PROPERTY NumOfHangers : DINT
GET
NumOfHangers:= SIf.Cur.dinNumOfHangersInBuffer;
END_GET
END_PROPERTY

METHOD PROTECTED sta_ERROR : BOOL
// state implemetation
//--------------------------------------------------------------------------------------
// Entry action
	IF (me.StateMachine.intState<>me.StateMachine.intStateLastCycle) THEN
		me.StateMachine.intStateHistory := me.StateMachine.intStateLastCycle; // -> possibillity to go back to state before error
		me.StateMachine.intStateLastCycle := me.StateMachine.intState;
		
	END_IF

//--------------------------------------------------------------------------------------
// Cyclic action
	IF (me.StateMachine.intState=me.StateMachine.intStateLastCycle) THEN
		
		// Switch valve off, cylinder back to extend position -> stop hanger
		SIf.Out.bolRetract.intern := FALSE;
		SIf.Out.bolRetract2.intern := TRUE;	
		
		// State Change Condition
		IF (CIf.Job.bolAlmReset = TRUE) THEN
			me.StateMachine.intStateNext := cSTA_ERRORQuit;
		END_IF
	END_IF

//--------------------------------------------------------------------------------------
// Exit action
	IF (me.StateMachine.intState<>me.StateMachine.intStateNext) THEN
		;
	END_IF
END_METHOD

METHOD PROTECTED sta_OFF : BOOL
// state implemetation
//--------------------------------------------------------------------------------------
// Entry action
	IF (me.StateMachine.intState<>me.StateMachine.intStateLastCycle) THEN
		me.StateMachine.intStateLastCycle := me.StateMachine.intState;
		
		// Reset total counter
		SIf.Cur.dinHangersPassedTotal:= 0;
	END_IF


//--------------------------------------------------------------------------------------
// Cyclic action
	IF (me.StateMachine.intState=me.StateMachine.intStateLastCycle) THEN
		
	
		// State Change Condition
		IF (me.Alarm.eActivAlmClass<>E_AlmClass.EOFF) AND (me.Alarm.eActivAlmClass<>E_AlmClass.OFF) THEN
			IF (me.intCmd=cCMD_STOP) THEN
				me.StateMachine.intStateNext :=  cSTA_STOPBusy;
			ELSIF (me.intCmd=STB_CmdState.cCMD_RELEASE) THEN 
				me.StateMachine.intStateNext := STB_CmdState.cSTA_RELEASEBusy;
			ELSIF(me.intCmd=STB_CmdState.cCMD_RELEASE_ALL) THEN
				me.StateMachine.intStateNext := STB_CmdState.cSTA_RELEASE_ALLBusy;
			ELSIF(me.intCmd=cCMD_RUN) THEN
				me.StateMachine.intStateNext := cSTA_RUNBusy;
			END_IF
		END_IF
	END_IF


//--------------------------------------------------------------------------------------
// Exit action
	IF (me.StateMachine.intState<>me.StateMachine.intStateNext) THEN
		;
	END_IF
END_METHOD

METHOD PROTECTED sta_OFFBusy : BOOL
// state implemetation
//--------------------------------------------------------------------------------------
// Entry action
	IF (me.StateMachine.intState<>me.StateMachine.intStateLastCycle) THEN
		me.StateMachine.intStateLastCycle := me.StateMachine.intState;
			
	END_IF

//--------------------------------------------------------------------------------------
// Cyclic action
	IF (me.StateMachine.intState=me.StateMachine.intStateLastCycle) THEN
		
		// Switch valve off, cylinder back to extend position -> stop hanger
		SIf.Out.bolRetract.intern := FALSE;
		SIf.Out.bolRetract2.intern := TRUE;	
			
		// State Change Condition
		IF (FALSE) THEN
			;
		ELSIF (TRUE) THEN
			me.StateMachine.intStateNext := cSTA_OFF;
		END_IF
	END_IF


//--------------------------------------------------------------------------------------
// Exit action
	IF (me.StateMachine.intState<>me.StateMachine.intStateNext) THEN
		;
	END_IF
END_METHOD

METHOD PROTECTED sta_RELEASE : BOOL
// state implemetation
//--------------------------------------------------------------------------------------
// Entry action
	IF (me.StateMachine.intState<>me.StateMachine.intStateLastCycle) THEN
		me.StateMachine.intStateLastCycle := me.StateMachine.intState;
			
		;
	END_IF

//--------------------------------------------------------------------------------------
// Cyclic action
	IF (me.StateMachine.intState=me.StateMachine.intStateLastCycle) THEN
		
		// Switch valve off, cylinder back to extend position -> stop hanger
		SIf.Out.bolRetract.intern := FALSE;
		SIf.Out.bolRetract2.intern := TRUE;	
		
		// State Change Condition
		IF (me.intCmd=cCMD_STOP) THEN
			me.StateMachine.intStateNext := cSTA_STOPBusy;
		ELSIF(me.intCmd=STB_CmdState.cCMD_RELEASE_ALL) THEN
			me.StateMachine.intStateNext := STB_CmdState.cSTA_RELEASE_ALLBusy;
		END_IF
		
	END_IF

//--------------------------------------------------------------------------------------
// Exit action
	IF (me.StateMachine.intState<>me.StateMachine.intStateNext) THEN
		;
	END_IF
END_METHOD

METHOD PROTECTED sta_RELEASE_ALL : BOOL
// state implemetation
//--------------------------------------------------------------------------------------
// Entry action
	IF (me.StateMachine.intState<>me.StateMachine.intStateLastCycle) THEN
		me.StateMachine.intStateLastCycle := me.StateMachine.intState;	
		;
	END_IF

//--------------------------------------------------------------------------------------
// Cyclic action
	IF (me.StateMachine.intState=me.StateMachine.intStateLastCycle) THEN
		

		// State Change Condition
		IF ((me.intCmd=cCMD_STOP) OR (me.intCmd=STB_CmdState.cCMD_RELEASE)) THEN
			me.StateMachine.intStateNext := cSTA_STOPBusy;
		END_IF
	END_IF

//--------------------------------------------------------------------------------------
// Exit action
	IF (me.StateMachine.intState<>me.StateMachine.intStateNext) THEN
		;
	END_IF
END_METHOD

METHOD PROTECTED sta_RELEASE_ALLBusy : BOOL
// state implemetation
//--------------------------------------------------------------------------------------
// Entry action
	IF (me.StateMachine.intState<>me.StateMachine.intStateLastCycle) THEN
		me.StateMachine.intStateLastCycle := me.StateMachine.intState;
				
		dinNumOfHangersToRelease:= 0;
		dinSetNumOfHangersToRelease:= 0;
		
		// Reset package counter
		SIf.Cur.dinHangersPassedPackage:= 0;
	
		// Initialize sub state machine
		me.SubStateMachine.intState:= cSTA_SUB_INITIALIZED; 
		me.SubStateMachine.intStateNext:= cSTA_SUB_INITIALIZED;
	
	END_IF

//--------------------------------------------------------------------------------------
// Cyclic action
	IF (me.StateMachine.intState=me.StateMachine.intStateLastCycle) THEN
			
		//--------------------------------------------------------------------------------------
		// sub state machine for release all sequence
		CASE me.SubStateMachine.intState OF
			//--------------------------------------------------------------------------------------
			cSTA_SUB_INITIALIZED:
				// Entry action
				IF (me.SubStateMachine.intState<>me.SubStateMachine.intStateLastCycle) THEN
					me.SubStateMachine.intStateLastCycle := me.SubStateMachine.intState;							
					
					//Used buffer mode?
					CASE SIf.Par.usiBuffermode OF
					0: // 0= Emptying buffer, use buffer capacity at cycle start
						dinSetNumOfHangersToRelease := SIf.Cfg.dinMaxCapacity;
					1: // 1= Emptying buffer, newly added hangers will be considered
						dinSetNumOfHangersToRelease := dinNumOfHangersToRelease;
					END_CASE
				
				END_IF
				
				// Simulation
				IF (CIf.SwCfg.bolSimulation) THEN
					;
				END_IF
	
				// State Change Condition
				IF(TRUE)THEN
					me.SubStateMachine.intStateNext := cSTA_SUB_HANGER_PASSING;
				END_IF
						
			//--------------------------------------------------------------------------------------
			cSTA_SUB_HANGER_PASSING:
				// Entry action
				IF (me.SubStateMachine.intState<>me.SubStateMachine.intStateLastCycle) THEN
					me.SubStateMachine.intStateLastCycle := me.SubStateMachine.intState;							
									
					// Check if min. one hanger exist and save info tmp. Used for counting.
					IF (SIf.In.bolHangerDetected.intern = TRUE) THEN
						bolHangerDetected:= TRUE;
					ELSE
						bolHangerDetected:= FALSE;
					END_IF
					
				END_IF
				
				// Simulation
				IF (CIf.SwCfg.bolSimulation) THEN
					;
				END_IF

				// Release all based on time and both pins go up or with pulses
				IF (SIf.Cfg.bolReleaseAllNonPulse = TRUE) THEN
					
					SIf.Out.bolRetract.intern := TRUE; // both pins move up
					SIf.Out.bolRetract2.intern := TRUE; // both pins move up
					
					// wait release all time
					IF (me.SubStateMachine.udiTimeInState_ms > SIf.Par.udiReleaseAllTime_ms) THEN
						me.SubStateMachine.intStateNext := cSTA_SUB_HANGER_PASSED;
					END_IF
					
					// Calculate number of hangers in buffer dependent number of hangers per pulse
					SIf.Cur.dinNumOfHangersInBuffer := 0;
					// Calculate total counter dependent number of hangers per pulse
					SIf.Cur.dinHangersPassedTotal:= SIf.Cur.dinHangersPassedTotal + dinNumOfHangersToRelease;
					// Calculate package counter dependent number of hangers per pulse				
					SIf.Cur.dinHangersPassedPackage:= SIf.Cur.dinHangersPassedPackage + dinNumOfHangersToRelease;
					// calculate hangers still to release
					dinSetNumOfHangersToRelease := 0;
					
				ELSE
					
					// Switch valve on, cylinder to retract position -> release hanger
					SIf.Out.bolRetract.intern := TRUE;  // pin move up
					SIf.Out.bolRetract2.intern := FALSE;  // pin move down
					
					// Pulse timer expired?
					IF (me.SubStateMachine.udiTimeInState_ms > SIf.Par.udiPulseLengthValve_ms) THEN
						me.SubStateMachine.intStateNext := cSTA_SUB_HANGER_PASSED;
						
						// Update all counters. Only if a hanger was detected before.
						// If no hanger detection sensor exists, count unconditional with every cylinder stroke
						IF (bolHangerDetected = TRUE) OR (Sif.Cfg.bolHasHangerDetection = FALSE) THEN
							
							// Note: Only for separator the number of hangers per pulse corresponds exactly the real number of passed hangers.
							// For all other units like e.g. double stopper it's only an approximate number.
						
							IF (SIf.Cfg.bolHasDecrementSensor = FALSE) THEN // Else do it in Method Always
								// Calculate number of hangers in buffer dependent number of hangers per pulse
								SIf.Cur.dinNumOfHangersInBuffer:= SIf.Cur.dinNumOfHangersInBuffer - dinNumOfHangersToRelease;
							END_IF
							// Calculate total counter dependent number of hangers per pulse
							SIf.Cur.dinHangersPassedTotal:= SIf.Cur.dinHangersPassedTotal + dinNumOfHangersToRelease;
							// Calculate package counter dependent number of hangers per pulse				
							SIf.Cur.dinHangersPassedPackage:= SIf.Cur.dinHangersPassedPackage + dinNumOfHangersToRelease;
							// calculate hangers still to release
							dinSetNumOfHangersToRelease := dinSetNumOfHangersToRelease - dinNumOfHangersToRelease;
							
							// Calculate NumOfHangersToRelease, Used for RELEASE_ALL end condition
							// Has buffer?
							// calculate max number of hangers could release per pulse
							IF (SIf.Cur.dinNumOfHangersInBuffer<=SIf.Cfg.uinNumOfHangersPerPulse) THEN
								dinNumOfHangersToRelease := SIf.Cur.dinNumOfHangersInBuffer;
							ELSE
								dinNumOfHangersToRelease := SIf.Cfg.uinNumOfHangersPerPulse;
							END_IF
							
							//Used buffer mode?
							CASE SIf.Par.usiBuffermode OF
								0:  
									IF  (dinNumOfHangersToRelease <= 0) THEN // All hangers should be released, do the hole capacity 
										dinSetNumOfHangersToRelease:= dinSetNumOfHangersToRelease - SIf.Cfg.uinNumOfHangersPerPulse;
									END_IF
								1:
									dinSetNumOfHangersToRelease:= dinNumOfHangersToRelease;
							END_CASE
													
							bolHangerDetected:= FALSE;
						END_IF
					END_IF
						
				END_IF
	
			//--------------------------------------------------------------------------------------
			cSTA_SUB_HANGER_PASSED:
				// Entry action
				IF (me.SubStateMachine.intState<>me.SubStateMachine.intStateLastCycle) THEN
					me.SubStateMachine.intStateLastCycle := me.SubStateMachine.intState;							
					;						
				END_IF
				
				// Switch valve off, cylinder back to extend position -> stop hanger
				SIf.Out.bolRetract.intern := FALSE;
				SIf.Out.bolRetract2.intern := TRUE;	
				
				// Simulation
				IF (CIf.SwCfg.bolSimulation) THEN
					;
				END_IF
					
				// State Change Condition
				IF ((dinSetNumOfHangersToRelease<=0) AND ((Sif.Cfg.bolHasHangerDetection = FALSE) OR (SIf.Par.usiBuffermode<>1))) THEN
					me.SubStateMachine.intStateNext := cSTA_SUB_FINISHED;
				ELSIF ((SIf.Par.usiBuffermode=1) AND (Sif.Cfg.bolHasHangerDetection = TRUE) AND (SIf.In.bolHangerDetected.intern = FALSE)) THEN
					me.SubStateMachine.intStateNext := cSTA_SUB_FINISHED;
				ELSIF (me.SubStateMachine.udiTimeInState_ms > SIf.Par.udiIntervalBufferEmptying_ms) THEN
					me.SubStateMachine.intStateNext := cSTA_SUB_HANGER_PASSING;
				END_IF
			
			//--------------------------------------------------------------------------------------
			cSTA_SUB_FINISHED:
					;	// Buffer emptied 
					
		END_CASE
			
		// State Change Condition
		// [ms] Timeout buffer emptying -> ERROR,(0 = disable monitoring)
		IF ((me.StateMachine.udiTimeInState_ms > (SIf.Par.udiTimeoutBufferEmptying_ms)) AND (SIf.Par.udiTimeoutBufferEmptying_ms <> 0)) THEN
			// SIf.Alm[1].strText := 'Timeout buffer emptying';
			pfbAlarmCtrl^.setAlarm(CIf.Info.intCtrlId,1,0,ADR(SIf.Alm),E_AlmState.RST,CIf.Job.eMe_ActivAlmClass);
			me.StateMachine.intStateNext := cSTA_ERROR;
		ELSIF (me.SubStateMachine.intState = cSTA_SUB_FINISHED) THEN				// Buffer emptied -> RELEASE_ALL
			me.StateMachine.intStateNext := STB_CmdState.cSTA_RELEASE_ALL;
		ELSIF(me.intCmd=cCMD_STOP) THEN
			me.StateMachine.intStateNext := cSTA_STOPBusy;		
		END_IF
	END_IF


//--------------------------------------------------------------------------------------
// Exit action
	IF (me.StateMachine.intState<>me.StateMachine.intStateNext) THEN
		;
	END_IF
END_METHOD

METHOD PROTECTED sta_RELEASEBusy : BOOL
// state implemetation
//--------------------------------------------------------------------------------------
// Entry action
	IF (me.StateMachine.intState<>me.StateMachine.intStateLastCycle) THEN
		me.StateMachine.intStateLastCycle := me.StateMachine.intState;

		// Check if min. one hanger exist and save info tmp. Used for counting in state RELEASE.	
		IF (SIf.In.bolHangerDetected.intern = TRUE) THEN
			bolHangerDetected:= TRUE;
		ELSE
			bolHangerDetected:= FALSE;
		END_IF
	
	END_IF

//--------------------------------------------------------------------------------------
// Cyclic action
	IF (me.StateMachine.intState=me.StateMachine.intStateLastCycle) THEN
		
		// Switch valve on, cylinder to retract position -> release hanger
		SIf.Out.bolRetract.intern := TRUE;
		SIf.Out.bolRetract2.intern := FALSE;	
		
		// State Change Condition
		IF (me.StateMachine.udiTimeInState_ms > SIf.Par.udiPulseLengthValve_ms) THEN
			me.StateMachine.intStateNext := STB_CmdState.cSTA_RELEASE;
	
			// Update all counters. Only if a hanger was detected before.
			// If no hanger detection sensor exists, count unconditional with every cylinder stroke
			IF (bolHangerDetected = TRUE) OR (SIf.Cfg.bolHasHangerDetection = FALSE) THEN
				
				// Note: Only for separator the number of hangers per pulse corresponds exactly the real number of passed hangers.
				// For all other units like e.g. double stopper it's only an approximate number.
			
				IF (SIf.Cfg.bolHasDecrementSensor = FALSE) THEN // Else do it in Method Always
					IF (SIf.Cfg.bolHasBufferFullSensor = TRUE AND SIf.In.bolBufferFull.intern = FALSE) THEN
						// Calculate number of hangers in buffer dependent number of hangers per pulse
						SIf.Cur.dinNumOfHangersInBuffer:= SIf.Cur.dinNumOfHangersInBuffer - dinNumOfHangersToRelease;
					ELSIF SIf.Cfg.bolHasBufferFullSensor = FALSE THEN
						// Calculate number of hangers in buffer dependent number of hangers per pulse
						SIf.Cur.dinNumOfHangersInBuffer:= SIf.Cur.dinNumOfHangersInBuffer - dinNumOfHangersToRelease;						
					END_IF
				END_IF
					
				// Calculate total counter dependent number of hangers per pulse
				SIf.Cur.dinHangersPassedTotal:= SIf.Cur.dinHangersPassedTotal + dinNumOfHangersToRelease;
				
				bolHangerDetected:= FALSE;
			END_IF
				
		END_IF
		
	END_IF

//--------------------------------------------------------------------------------------
// Exit action
	IF (me.StateMachine.intState<>me.StateMachine.intStateNext) THEN
		;
	END_IF
END_METHOD

METHOD PROTECTED sta_RUN : BOOL
// state implemetation
//--------------------------------------------------------------------------------------
// Entry action
	IF (me.StateMachine.intState<>me.StateMachine.intStateLastCycle) THEN
		me.StateMachine.intStateLastCycle := me.StateMachine.intState;
		
		// Init sub state machine	
		me.SubStateMachine.intState := cSTA_SUB_CHECK_FOR_RESERVATION; 
		me.SubStateMachine.intStateNext := cSTA_SUB_CHECK_FOR_RESERVATION; 
	END_IF

//--------------------------------------------------------------------------------------
// Cyclic action
	IF (me.StateMachine.intState=me.StateMachine.intStateLastCycle) THEN
		
		//----------------------------------------------------------------------
		// Calculate position for transport 
		//----------------------------------------------------------------------	
		// If this task is in faster cycle then the parent, calculate internal position more exactly during the taskcycle
		IF dinTransportPositionOld_um <> SIf.Cur.dinTransportPosition_um THEN
			SIf.Cur.dinTransportPositionCalc_um := SIf.Cur.dinTransportPosition_um;
			dinTransportPositionOld_um := SIf.Cur.dinTransportPosition_um;
			dinPositionCorrection_um := 0;
		ELSE
			dinPositionCorrection_um := dinPositionCorrection_um + LREAL_TO_DINT(DINT_TO_LREAL(SIf.Cur.dinTransportspeed_um_s) * UDINT_TO_LREAL(me.FUBInfo.udiSample_ms) / 1000.0 );
			SIf.Cur.dinTransportPositionCalc_um := dinTransportPositionOld_um + dinPositionCorrection_um;
		END_IF
				
		//--------------------------------------------------------------------------------------
		// sub state machine
		CASE me.SubStateMachine.intState OF
			//--------------------------------------------------------------------------------------
			cSTA_SUB_CHECK_FOR_RESERVATION:
			
				IF (me.SubStateMachine.intState<>me.SubStateMachine.intStateLastCycle) THEN
					me.SubStateMachine.intStateLastCycle := me.SubStateMachine.intState;
					;
				END_IF
			
				// Simulation
				IF (CIf.SwCfg.bolSimulation) THEN
					;
				END_IF
							
				// Calculate trigger "negative" position offset.
				// Note: The trigger offset must be calculated dependent the drive (transport) speed 
				// Formular: TrigNegPosOffset = DriveSpeed * TimeOnSlide	
				dinCalcTrigNegPosOffset_um:= REAL_TO_DINT (DINT_TO_REAL(SIf.Cur.dinTransportspeed_um_s) * (UINT_TO_REAL(SIf.Par.uinTimeOnSlide_ms) / 1000));
					
				// Check trigger window
				FOR intBufferIndex := 0 TO Const_MTR.cusiSectionBuffer_SIZE DO
					// Check if the current transport position is within the trigger window and if section is reserved for this instance to release the hanger
					IF ((SIf.Par.dinPositionOfSlide_um < (SIf.Cur.pSectionBuffer^[intBufferIndex].dinTrigStartPos - dinCalcTrigNegPosOffset_um))
						AND (SIf.Par.dinPositionOfSlide_um > (SIf.Cur.pSectionBuffer^[intBufferIndex].dinTrigEndPos - dinCalcTrigNegPosOffset_um))
						AND (SIf.Cur.pSectionBuffer^[intBufferIndex].enmState = E_Typ_MTR_SECTION_STATE.Reserved) AND (SIf.Cur.pSectionBuffer^[intBufferIndex].usiReservedForLine = SIf.Cfg.usiLineNumber)) THEN						
							// Section is free and reserved for this instance -> hanger can be released!
							// Update status for the section
							SIf.Cur.pSectionBuffer^[intBufferIndex].enmState := E_Typ_MTR_SECTION_STATE.HangerOnSlide;
							me.SubStateMachine.intStateNext := cSTA_SUB_RELEASE_BUSY;
							EXIT;
					END_IF
				END_FOR					
				
			//--------------------------------------------------------------------------------------
			cSTA_SUB_RELEASE_BUSY:
				IF (me.SubStateMachine.intState<>me.SubStateMachine.intStateLastCycle) THEN
					me.SubStateMachine.intStateLastCycle := me.SubStateMachine.intState;
					;
				END_IF
			
				// Switch valve on, cylinder to retract position -> release hanger
				SIf.Out.bolRetract.intern := TRUE;
				
				// State Change Condition
				IF (me.SubStateMachine.udiTimeInState_ms > SIf.Par.udiPulseLengthValve_ms) THEN
					// Next step
					me.SubStateMachine.intStateNext := cSTA_SUB_STOP;
			
					// Update all counters. Only if a hanger was detected before.
					// If no hanger detection sensor exists, count unconditional with every cylinder stroke
					IF (SIf.In.bolHangerDetected.intern = TRUE) OR (SIf.Cfg.bolHasHangerDetection = FALSE) THEN
						
						// Note: Only for separator the number of hangers per pulse corresponds exactly the real number of passed hangers.
						// For all other units like e.g. double stopper it's only an approximate number.
					
						IF (SIf.Cfg.bolHasDecrementSensor = FALSE) THEN // Else do it in Method Always
							IF (SIf.Cfg.bolHasBufferFullSensor = TRUE AND SIf.In.bolBufferFull.intern = FALSE) THEN
								// Calculate number of hangers in buffer dependent number of hangers per pulse
								SIf.Cur.dinNumOfHangersInBuffer:= SIf.Cur.dinNumOfHangersInBuffer - dinNumOfHangersToRelease;
							ELSIF SIf.Cfg.bolHasBufferFullSensor = FALSE THEN
								// Calculate number of hangers in buffer dependent number of hangers per pulse
								SIf.Cur.dinNumOfHangersInBuffer:= SIf.Cur.dinNumOfHangersInBuffer - dinNumOfHangersToRelease;						
							END_IF
						END_IF						
						// Calculate total counter dependent number of hangers per pulse
						SIf.Cur.dinHangersPassedTotal:= SIf.Cur.dinHangersPassedTotal + dinNumOfHangersToRelease;		
					END_IF
						
				END_IF
			
			//--------------------------------------------------------------------------------------
			cSTA_SUB_STOP:
				IF (me.SubStateMachine.intState<>me.SubStateMachine.intStateLastCycle) THEN
					me.SubStateMachine.intStateLastCycle := me.SubStateMachine.intState;
				END_IF
				
				// Update status for the section
				SIf.Cur.pSectionBuffer^[intBufferIndex].enmState := E_Typ_MTR_SECTION_STATE.HangerReleased;
				// Switch valve off, cylinder back to extend position -> stop hanger
				SIf.Out.bolRetract.intern := FALSE;
			
				// State Change Condition
				// Check error if retracted position not reached
				IF (TRUE) THEN
					me.SubStateMachine.intStateNext := cSTA_SUB_CHECK_FOR_RESERVATION;
				END_IF
		
			
		END_CASE
		
		// State Change Condition
		IF(me.intCmd=cCMD_STOP) THEN
			me.StateMachine.intStateNext := cSTA_STOPBusy;	
		END_IF
		
	END_IF

//--------------------------------------------------------------------------------------
// Exit action
	IF (me.StateMachine.intState<>me.StateMachine.intStateNext) THEN
	;
	END_IF
END_METHOD

METHOD PROTECTED sta_RUNBusy : BOOL
// state implemetation
//--------------------------------------------------------------------------------------
// Entry action
	IF (me.StateMachine.intState<>me.StateMachine.intStateLastCycle) THEN
		me.StateMachine.intStateLastCycle := me.StateMachine.intState;
		;				
	END_IF

//--------------------------------------------------------------------------------------
// Cyclic action
	IF (me.StateMachine.intState=me.StateMachine.intStateLastCycle) THEN
			
		// State Change Condition
		
		// Check if access to section buffer exist. 
		// This controller will be set to RUN in case if STB work in combination with FUB MTR to merge hangers into a TLK.
		IF (SIf.Cur.pSectionBuffer = 0) THEN
			// SIf.Alm[4].strText := 'RUN not possible, no access to section buffer';
			pfbAlarmCtrl^.setAlarm(CIf.Info.intCtrlId,4,0,ADR(SIf.Alm),E_AlmState.RST,CIf.Job.eMe_ActivAlmClass);	
			me.StateMachine.intStateNext := cSTA_ERROR;
		ELSE
			me.StateMachine.intStateNext := cSTA_RUN;		
		END_IF
	END_IF

//--------------------------------------------------------------------------------------
// Exit action
	IF (me.StateMachine.intState<>me.StateMachine.intStateNext) THEN
		;
	END_IF
END_METHOD

METHOD PROTECTED sta_STOP : BOOL
// state implemetation
//--------------------------------------------------------------------------------------
// Entry action
	IF (me.StateMachine.intState<>me.StateMachine.intStateLastCycle) THEN
		me.StateMachine.intStateLastCycle := me.StateMachine.intState;
		
		bolErrorPosLost:= FALSE;
		uinPosEdgeCounter:= 0;
	END_IF


//--------------------------------------------------------------------------------------
// Cyclic action
	IF (me.StateMachine.intState=me.StateMachine.intStateLastCycle) THEN
	
		//--------------------------------------------------------------------
		// Monitoring for cylinder position lost
		//--------------------------------------------------------------------
		IF (Sif.cfg.bolCylPosLostMonitoring=TRUE) THEN
			
			// -> Checked indirectly via sensor "buffer full" or "hanger detected" if exist.
			
			// Decision, which sensor should be used for monitoring
			// Prio 1. Always use the hanger detection sensor if exists
			IF (SIf.Cfg.bolHasHangerDetection = TRUE) THEN
				// Use hanger detection sensor signal
				bolSignalForPosLostMonitoring:= SIf.In.bolHangerDetected.intern;
			ELSE
				// Prio 2. Check if buffer full sensor exists 
				IF (SIf.Cfg.bolHasBufferFullSensor = TRUE) THEN
					// Use buffer full sensor signal
					bolSignalForPosLostMonitoring:= SIf.In.bolBufferFull.intern;
				ELSE
					// No sensor exist. Not possible to monitor cylinder position lost! 
					bolSignalForPosLostMonitoring:= FALSE;
				END_IF
			END_IF
				
			// Count sensor pos. edges
			IF ((bolSignalForPosLostMonitoring <> bolSignalForPosLostMonitoringOld) AND (bolSignalForPosLostMonitoring = TRUE))THEN	
				uinPosEdgeCounter:= uinPosEdgeCounter + 1;
			END_IF
			bolSignalForPosLostMonitoringOld:= bolSignalForPosLostMonitoring;
						
			// Check condition for set error
			// Wait until the counter is > than dinMaxNumOfHangers_PosMonitoring
			IF (uinPosEdgeCounter > SIf.Cfg.dinMaxNumOfHangers_PosMonitoring) THEN
				bolErrorPosLost:= TRUE;
			END_IF
			
		END_IF
		
		//--------------------------------------------------------------------
		//--------------------------------------------------------------------
		
		// State Change Condition	
		// Error cylinder position lost
		IF ((bolErrorPosLost=TRUE) AND (Sif.cfg.bolCylPosLostMonitoring=TRUE))THEN
			// SIf.Alm[3].strText := 'Cylinder position lost. Hangers slip through';
			pfbAlarmCtrl^.setAlarm(CIf.Info.intCtrlId,3,0,ADR(SIf.Alm),E_AlmState.RST,CIf.Job.eMe_ActivAlmClass);
			bolErrorPosLost:= FALSE;
			uinPosEdgeCounter:= 0;
			me.StateMachine.intStateNext := cSTA_ERROR;
		ELSIF (me.intCmd=STB_CmdState.cCMD_RELEASE) THEN 
			me.StateMachine.intStateNext := STB_CmdState.cSTA_RELEASEBusy;
		ELSIF(me.intCmd=STB_CmdState.cCMD_RELEASE_ALL) THEN
			me.StateMachine.intStateNext := STB_CmdState.cSTA_RELEASE_ALLBusy;
		ELSIF (me.intCmd=cCMD_RUN) THEN
			me.StateMachine.intStateNext := cSTA_RUNBusy;
		END_IF
	END_IF

//-------------------------------------------------------------------------------------
// Exit action
	IF (me.StateMachine.intState<>me.StateMachine.intStateNext) THEN
		;
	END_IF
END_METHOD

METHOD PROTECTED sta_STOPBusy : BOOL
// state implemetation
//--------------------------------------------------------------------------------------
// Entry action
	IF (me.StateMachine.intState<>me.StateMachine.intStateLastCycle) THEN
		me.StateMachine.intStateLastCycle := me.StateMachine.intState;

	END_IF


//--------------------------------------------------------------------------------------
// Cyclic action
	IF (me.StateMachine.intState=me.StateMachine.intStateLastCycle) THEN
			
		// Switch valve off, cylinder back to extend position -> stop hanger
		SIf.Out.bolRetract.intern := FALSE;
		SIf.Out.bolRetract2.intern := TRUE;	
				
		// State Change Condition
		IF (me.StateMachine.udiTimeInState_ms > SIf.Par.udiPulseLengthValve_ms) THEN
			me.StateMachine.intStateNext := cSTA_STOP;
		END_IF
	END_IF


//--------------------------------------------------------------------------------------
// Exit action
	IF (me.StateMachine.intState<>me.StateMachine.intStateNext) THEN
		;
	END_IF
END_METHOD

METHOD PROTECTED StateMachine : BOOL
SUPER^.StateMachine();

// main statemachine of base controller
CASE me.StateMachine.intState OF
	cSTA_RUNBusy: 
        THIS^.sta_RUNBusy();
    cSTA_RUN: 
        THIS^.sta_RUN();
    cSTA_STOPBusy: 
        THIS^.sta_STOPBusy();
    cSTA_STOP: 
        THIS^.sta_STOP();
    STB_CmdState.cSTA_RELEASE_ALLBusy: 
        THIS^.sta_RELEASE_ALLBusy();
    STB_CmdState.cSTA_RELEASE_ALL: 
        THIS^.sta_RELEASE_ALL();
    STB_CmdState.cSTA_RELEASEBusy: 
        THIS^.sta_RELEASEBusy();
    STB_CmdState.cSTA_RELEASE: 
        THIS^.sta_RELEASE();
END_CASE;
END_METHOD

END_FUNCTION_BLOCK

// POUs/Controller/Lvl2/MTR (Merger Transport)/FB_MTR
FUNCTION_BLOCK FB_MTR EXTENDS FB_CtrlBase IMPLEMENTS IBuffer
VAR_INPUT
	/// Sensor hanger detected
	In_bolHangerDetected: BOOL;
	/// Sensor pin detected
	In_bolPinDetected: BOOL;
END_VAR
VAR
	/// Specific interface struct for public access
	SIf: T_Ctrl_SIf_MTR;
	/// Section buffer
	a_stSectionBuffer: ARRAY[0..Const_MTR.cusiSectionBuffer_SIZE] OF T_MTR_Buffer_Sections;
	/// List of pointers to Childs
	a_pLineChildCtrl: ARRAY[0..Base_Const.cMaxNrOfChilds] OF POINTER TO FB_STB;
	/// List of childs common interface
	a_pLineChildCIF: ARRAY[0..Base_Const.cMaxNrOfChilds] OF POINTER TO T_Ctrl_CIf;
	/// List of childs specific interface for additional parameters or cur
	a_pLineChildSIF: ARRAY[0..Base_Const.cMaxNrOfChilds] OF POINTER TO T_Ctrl_SIf_STB;
	usiNumOfLines: USINT;
	usiNumOfValidPointerToLine: USINT;
	/// Last new position value from parent
	dinTransportPositionOld_um: DINT;
	/// Driven Way in the task
	dinDrivenWay_um: DINT;
	/// Position correction in faster Task cycletime
	dinPositionCorrection_um: DINT;
	/// Edge detection of the inputs
	bolRE_HangerDetected: BOOL;
	bolRE_PinDetected: BOOL;
	/// Position of the last line. Used to detect if a section is driven out
	dinPositionOfLastLine_um: DINT;
	/// Loop variable
	intLine: INT;
	bolExit: BOOL;
	/// Simulated section length
	dinSimSectionLength_um: DINT := 510000;
	/// Simulated way to trigger section start/end
	dinSimWayTrigSection_um: DINT;
END_VAR

(*__________________________________________________________________________________________________
¦	
¦	Vistaprint Schweiz GmbH
¦	CH - 8401 Winterthur
¦
¦	www.vistaprint.ch - info@vistaprint.ch
¦___________________________________________________________________________________________________

Function desription:
This controller will be used in combination with childs of type STB to merge hangers
from different slides into a transport system of type TLK.

History:
Version		Date			Author		Comment
---------------------------------------------------------------------------------------------------
0.00.1		25.04.2014		AVME/DSC	Start history.				  
								
__________________________________________________________________________________________________*)


IF ((me.bolActivate) AND (THIS^.checkChildValid())) THEN // cyclic call enabled
	IF (CIf.Info.bolInitDone=FALSE) THEN // first cycle -> init
		CtrlInit();
		CIf.Info.bolInitDone := TRUE;
	ELSE
		CycleStartDuty();
	
		Always();
		
		StateMachine();
		
		CycleEndDuty();
	END_IF
END_IF;

METHOD AddLine
VAR_INPUT
	p_Line: POINTER TO FB_STB;
END_VAR

// Method add the pointer address of the line child controller to the array list.
IF (usiNumOfLines <= (Base_Const.cMaxNrOfChilds-1)) THEN
	// Add line child controller to list
	a_pLineChildCtrl[usiNumOfLines] := p_Line;
	// Inc. number of lines
	usiNumOfLines:= usiNumOfLines+1;
	// Check if the pointer is valid
	IF (p_Line<>0) THEN
		usiNumOfValidPointerToLine:= usiNumOfValidPointerToLine+1;
	END_IF
END_IF
END_METHOD

METHOD PROTECTED Always : BOOL
VAR
	ii: INT;
END_VAR
IF (me.bolChangeBackToAUTO=TRUE) THEN // switch mode to automatic switch off controller
	//me.StateMachine.intStateNext := cSTA_OFFBusy;
	//me.bolChangeBackToAUTO := FALSE; // for cylinder no change to off when switch to automatic!!
END_IF

SUPER^.Always();

// ----------------------------------------------------------------------------------
// cyclic actions outside of statemachine
IF (me.StateMachine.intState<>cSTA_SINGLE_ANSWER) THEN
	
	//-------------------------------------------------
	// Provide current values for the parent
	//-------------------------------------------------	
	
	// Number of lines to merge, depends on how many times the method "AddLine" was called at init
	SIf.Cur.usiNumOfLinesToMerge:= usiNumOfLines;
	// Actual Item Count of this controller -> based on all lines
	SIf.Cur.dinCurrentItemCount:= THIS^.CalcSumOfItems();
	// Max. buffer capacity -> based on all lines
	SIf.Cur.dinMaxCapacity:= THIS^.CalcMaxCapacity();	

	//----------------------------------------------------------------------
	// Calculate position for transport 
	//----------------------------------------------------------------------
		
	// If this task is used in a faster cycle as the parent, the driven way will be indirectly calculated (synchronized) over the transport speed.
	// If transport position changed from the parent (new value), synchronize the driven way 
	
	IF (dinTransportPositionOld_um <> SIf.Cur.dinTransportPosition_um) THEN
		dinDrivenWay_um := SIf.Cur.dinTransportPosition_um - SIf.Cur.dinTransportPositionCalc_um;
		SIf.Cur.dinTransportPositionCalc_um := SIf.Cur.dinTransportPosition_um;
		dinTransportPositionOld_um := SIf.Cur.dinTransportPosition_um;
		dinPositionCorrection_um := 0;
	ELSE
		// During the time, if there is no position change from the parent, calculate the driven way dependent the speed of transport.		
		// s = v * t
		dinDrivenWay_um := LREAL_TO_DINT(DINT_TO_LREAL(SIf.Cur.dinTransportspeed_um_s) * UDINT_TO_LREAL(me.FUBInfo.udiSample_ms) / 1000.0 );
		dinPositionCorrection_um := dinPositionCorrection_um + dinDrivenWay_um;
		SIf.Cur.dinTransportPositionCalc_um := dinTransportPositionOld_um + dinPositionCorrection_um;
	END_IF
	
	//----------------------------------------------------------------------
	// Update transport position and speed to childs 
	//----------------------------------------------------------------------
	FOR ii:=0 TO usiNumOfLines-1 BY 1 DO	
		a_pLineChildSIF[ii]^.Cur.dinTransportPosition_um := SIf.Cur.dinTransportPosition_um;
		a_pLineChildSIF[ii]^.Cur.dinTransportspeed_um_s := SIf.Cur.dinTransportspeed_um_s;
	END_FOR

END_IF

// ----------------------------------------------------------------------------------
// Always change actions in Base Library
// ----------------------------------------------------------------------------------
// overrule error always from base -> no EOFF State!! in EOFF go to OFF
IF (me.StateMachine.intStateNext = cSTA_EOFFBusy) THEN
	IF (me.StateMachine.intState=cSTA_OFF) THEN
		me.StateMachine.intStateNext := cSTA_OFF;
	ELSE // stay in OFF
		me.StateMachine.intStateNext := cSTA_OFFBusy;
	END_IF
END_IF

// Conditions Always
IF (((me.Alarm.eActivAlmClass=E_AlmClass.EOFF) OR (me.Alarm.eActivAlmClass=E_AlmClass.OFF) OR (me.intCmd=cCMD_OFF))
		 AND (me.StateMachine.intState<>cSTA_ERROR) AND (me.StateMachine.intState<>cSTA_ERRORQuit) AND
		(me.StateMachine.intState<>cSTA_OFF) AND (me.StateMachine.intState<>cSTA_OFFBusy)) THEN
	// alarm evt EOFF, OFF or cmd off
	me.StateMachine.intStateNext := cSTA_OFFBusy;
END_IF
END_METHOD

PROPERTY BufferFull : BOOL
GET
BufferFull:= False;
END_GET
END_PROPERTY

METHOD PROTECTED CalcMaxCapacity : DINT
VAR
	ii: INT;
	dinSumMaxCapacity: DINT;
END_VAR
// Method calculate the sum of max. capacities from all lines and return the result.

//Init
CalcMaxCapacity:= 0;
dinSumMaxCapacity:= 0;

// Loop over all childs
FOR ii:=0 TO usiNumOfLines-1 BY 1 DO
	// Build sum of all lines		
	dinSumMaxCapacity:= dinSumMaxCapacity + a_pLineChildSIF[ii]^.Cfg.dinMaxCapacity; 	
END_FOR

// Return result
CalcMaxCapacity:= dinSumMaxCapacity;
END_METHOD

METHOD PROTECTED CalcSumOfItems : DINT
VAR
	ii: INT;
	dinSumOfItems: DINT;
END_VAR
// Method calculate the sum of hangers from all lines and return the result.

//Init
CalcSumOfItems:= 0;
dinSumOfItems:= 0;

// Loop over all childs
FOR ii:=0 TO usiNumOfLines-1 BY 1 DO
	// Build sum of all zones		
	dinSumOfItems:= dinSumOfItems + a_pLineChildSIF[ii]^.Cur.dinNumOfHangersInBuffer; 	
END_FOR

// Return result
CalcSumOfItems:= dinSumOfItems;
END_METHOD

METHOD checkChildAlmClass : BOOL
//------------------------------------------------------------------------------------------------------
// check child alarm classes
// set me alarm class active if at least one child has an EOFF
IF CheckAllChildAlmClass(E_AlmClass.EOFF) THEN
	CIf.Job.eMe_ActivAlmClass := E_AlmClass.EOFF;
	me.Alarm.bolfp := TRUE;
ELSIF CheckAllChildAlmClass(E_AlmClass.OFF) THEN
	CIf.Job.eMe_ActivAlmClass := E_AlmClass.OFF;
	me.Alarm.bolfp := TRUE;
ELSIF CheckAllChildAlmClass(E_AlmClass.STOP) THEN  // FB_MER needs alarm class STOP
	CIf.Job.eMe_ActivAlmClass := E_AlmClass.STOP;
	me.Alarm.bolfp := TRUE;
ELSE
	IF (me.Alarm.bolfp) THEN
		CIf.Job.eMe_ActivAlmClass := E_AlmClass.NONE; // no reset necessary
		me.Alarm.bolfp := FALSE;
	END_IF
END_IF

//------------------------------------------------------------------------------------------------------
// set alarm class parent of childs
//------------------------------------------------------------------------------------------------------
// set alarm class parent of childs in the case of a parent EOFF or me=OFF or EOFF
IF (CIf.Job.eParent_ActivAlmClass=E_AlmClass.EOFF) THEN
	SetAllChildAlmClass(CIf.Job.eParent_ActivAlmClass);
ELSIF(CIf.Job.eMe_ActivAlmClass=E_AlmClass.EOFF) OR (CIf.Job.eMe_ActivAlmClass=E_AlmClass.OFF) THEN
	SetAllChildAlmClass(CIf.Job.eMe_ActivAlmClass);
ELSE
	// no important alarm for child active
	SetAllChildAlmClass(E_AlmClass.NONE);
END_IF
END_METHOD

METHOD PROTECTED checkChildValid : BOOL
IF (usiNumOfLines = usiNumOfValidPointerToLine) THEN
	checkChildValid:= TRUE;
ELSE
	checkChildValid:= FALSE;
	// Invalid child pointer
	IF (usiNumOfLines <> usiNumOfValidPointerToLine) THEN
		// SIf.Alm[1].strText := 'Invalid child pointer'; 
		pfbAlarmCtrl^.setAlarm(CIf.Info.intCtrlId,1,0,ADR(SIf.Alm),E_AlmState.RST,CIf.Job.eMe_ActivAlmClass);	
	END_IF
END_IF
END_METHOD

METHOD PROTECTED checkStateAllLines : BOOL
VAR_INPUT
	cSTA: INT;
END_VAR
VAR
	ii: INT;
	usiNumOfCheckedChilds: USINT;
END_VAR
// Method check input state of all lines

//Init
checkStateAllLines:= FALSE;
usiNumOfCheckedChilds:= 0;

// Loop over all childs
FOR ii:=0 TO usiNumOfLines-1 BY 1 DO
	// Check state	
	// Special condition: In case if the child is in state ERROR and STOP is requested. Set child as checked.
	// Parent controller need state STOP that automatic stop sequence can work for all other childs.
	IF (a_pLineChildCIF[ii]^.Job.intState = cSTA) OR ((a_pLineChildCIF[ii]^.Job.intState = cSTA_ERROR) AND (cSTA = cSTA_STOP)) THEN
		usiNumOfCheckedChilds:= usiNumOfCheckedChilds+1;
		SIf.Cur.a_bolChildReady[ii] := TRUE;
	ELSE
		SIf.Cur.a_bolChildReady[ii] := FALSE;		
	END_IF

END_FOR

// All states equal the input state
IF (usiNumOfCheckedChilds = usiNumOfLines) THEN
	checkStateAllLines:= TRUE;
END_IF
END_METHOD

METHOD PROTECTED CmdToAllLines
VAR_INPUT
	cCMD: INT;
END_VAR
VAR
	ii: INT;
END_VAR
// Method send input command to all existing line child controller.
FOR ii:=0 TO usiNumOfLines-1 BY 1 DO	
	a_pLineChildCIF[ii]^.Job.intACmd:= cCMD;
END_FOR
END_METHOD

METHOD PROTECTED CtrlInit : BOOL
VAR
	ii: INT;
END_VAR
SUPER^.CtrlInit();

//----------------------------------------------------------------------
// Initialize all lines
//----------------------------------------------------------------------

// Method initialize all line child controller.
FOR ii:=0 TO usiNumOfLines-1 BY 1 DO	
	a_pLineChildCIF[ii] := THIS^.AddChild(a_pLineChildCtrl[ii]^);
	a_pLineChildSIF[ii] := a_pLineChildCtrl[ii]^.getCtrlSIf();
	// Initialize access from STB to section buffer
	a_pLineChildSIF[ii]^.Cur.pSectionBuffer := ADR(a_stSectionBuffer[0]);
END_FOR

//----------------------------------------------------------------------
// Determine position of the last line (slide)
//----------------------------------------------------------------------
dinPositionOfLastLine_um:= a_pLineChildSIF[usiNumOfLines-1]^.Par.dinPositionOfSlide_um;
END_METHOD

METHOD FB_init : BOOL
VAR_INPUT
	///if TRUE, the retain variables are initialized (warm start / cold start)
	bInitRetains: BOOL;
	///if TRUE, the instance afterwards gets moved into the copy code (online change)
	bInCopyCode: BOOL;
END_VAR
VAR
	ii: UINT;
END_VAR
//------------------------------------------------------------------------------------------------------------------------
// to manually change in new FUB implementation!!!
// define valid commands for this controller
FOR ii:= 0 TO (SIZEOF(CIf.Job.aCmdList)/SIZEOF(CIf.Job.aCmdList[0])-1) BY 1 DO
	IF (CIf.Job.aCmdList[ii].intCmd=cCMD_INITIALIZED) THEN
		// found first empty array element
		EXIT;
	END_IF
END_FOR

CIf.Job.aCmdList[ii].intCmd := cCMD_STOP;
CIf.Job.aCmdList[ii].strName := 'Stop'; 
CIf.Job.aCmdList[ii].bolAvailable := TRUE;
ii := ii +1;
CIf.Job.aCmdList[ii].intCmd := cCMD_RUN;
CIf.Job.aCmdList[ii].strName := 'Run';
CIf.Job.aCmdList[ii].bolAvailable := TRUE;

// set name of class/typ
CIf.Info.strType := 'FB_MTR'; 

// set alarm class
SIf.Alm[1].eAlmClass := E_AlmClass.STOP;
SIf.Alm[1].strText := 'Invalid child pointer';


//*******************************************************************************
// initial values
//*******************************************************************************

// software configuration
CIf.SwCfg.bolExist := TRUE;
CIf.SwCfg.bolSimulation := FALSE;

// configuration

// parameter
END_METHOD

METHOD getCtrlSIf : POINTER TO T_Ctrl_SIf_MTR
getCtrlSIf := ADR(SIf);
END_METHOD

METHOD PROTECTED IoInBridge : BOOL
// digitale and analoge inputs read from hardware or forcing
SIf.In.bolHangerDetected.map := THIS^.In_bolHangerDetected;
SIf.In.bolPinDetected.map := THIS^.In_bolPinDetected;

IF (CIf.SwCfg.bolSimulation = FALSE) THEN
	getInBol(CIf.Job.bolIoForce,ADR(SIf.In.bolHangerDetected));
	getInBol(CIf.Job.bolIoForce,ADR(SIf.In.bolPinDetected));
ELSE
	//simulation of global IO
END_IF
END_METHOD

PROPERTY MaxCapacity : DINT
GET
MaxCapacity:= SIf.Cur.dinMaxCapacity;
END_GET
END_PROPERTY

PROPERTY NumOfHangers : DINT
GET
NumOfHangers:= SIf.Cur.dinCurrentItemCount;
END_GET
END_PROPERTY

METHOD PROTECTED sta_OFF : BOOL
// state implemetation
//--------------------------------------------------------------------------------------
// Entry action
	IF (me.StateMachine.intState<>me.StateMachine.intStateLastCycle) THEN
		me.StateMachine.intStateLastCycle := me.StateMachine.intState;
		;		
	END_IF

//--------------------------------------------------------------------------------------
// Cyclic action
	IF (me.StateMachine.intState=me.StateMachine.intStateLastCycle) THEN
		
		// Reset total counter
		SIf.Cur.dinNumOfMergedHangersTotal:= 0;
		
		// State Change Condition
		IF (me.Alarm.eActivAlmClass<>E_AlmClass.EOFF) AND (me.Alarm.eActivAlmClass<>E_AlmClass.OFF) THEN
			IF (me.intCmd=cCMD_STOP) THEN
				me.StateMachine.intStateNext := cSTA_STOPBusy;
			ELSIF (me.intCmd=cCMD_RUN) THEN 
				me.StateMachine.intStateNext := cSTA_RUNBusy;
			END_IF
		END_IF
	END_IF

//--------------------------------------------------------------------------------------
// Exit action
	IF (me.StateMachine.intState<>me.StateMachine.intStateNext) THEN
		;
	END_IF
END_METHOD

METHOD PROTECTED sta_RUN : BOOL
VAR
	/// Looping variable
	intSec: INT;
	intDeleteRes: INT;
	intReservationCount: INT;
	intLineNum: INT;
END_VAR
// state implemetation
//--------------------------------------------------------------------------------------
// Entry action
	IF (me.StateMachine.intState<>me.StateMachine.intStateLastCycle) THEN
		me.StateMachine.intStateLastCycle := me.StateMachine.intState;	
		// Init	
		intLine:= 0;
	END_IF

//--------------------------------------------------------------------------------------
// Cyclic action
	IF (me.StateMachine.intState=me.StateMachine.intStateLastCycle) THEN
						
		//----------------------------------------------------------------------
		// Set the section start and end positions (triggered by pin sensor)
		//----------------------------------------------------------------------
		
		// Simulation of section start and end
		IF (CIf.SwCfg.bolSimulation = TRUE) THEN		
			SIf.In.bolPinDetected.intern:= FALSE;
			
			IF (dinSimWayTrigSection_um >= dinSimSectionLength_um) THEN
				dinSimWayTrigSection_um:= 0;
				// Set true for one cycle
				SIf.In.bolPinDetected.intern:= TRUE;
			END_IF
			// Increase position		
			dinSimWayTrigSection_um:= dinSimWayTrigSection_um + dinDrivenWay_um;				
		END_IF
				
		// Wait for positive edge of the pin sensor (pin detected)
		IF (SIf.In.bolPinDetected.intern = TRUE) AND (bolRE_PinDetected = FALSE) THEN
			bolRE_PinDetected := TRUE;
				
			// Loop over section buffer
			FOR intSec := 0 TO Const_MTR.cusiSectionBuffer_SIZE DO
				
				// If start position already set
				IF (a_stSectionBuffer[intSec].enmState = E_Typ_MTR_SECTION_STATE.StartPositionSet) THEN						
					// Set end position of the section
					a_stSectionBuffer[intSec].dinSecEndPos:= 0 - SIf.Par.dinPinLenght_um;
					a_stSectionBuffer[intSec].usiReservedForLine:= 0;
					a_stSectionBuffer[intSec].enmState:= E_Typ_MTR_SECTION_STATE.EndPositionSet;
				END_IF
				
				// Free buffer element  
				IF ((a_stSectionBuffer[intSec].enmState = E_Typ_MTR_SECTION_STATE.Undefined) OR (a_stSectionBuffer[intSec].enmState = E_Typ_MTR_SECTION_STATE.HangerReleased)) THEN			
					// Set start position of the section
					a_stSectionBuffer[intSec].dinSecStartPos:= 0 - SIf.Par.dinPinLenght_um;
					a_stSectionBuffer[intSec].enmState:= E_Typ_MTR_SECTION_STATE.StartPositionSet;
					EXIT;									  
				END_IF
												
			END_FOR
				
		ELSIF (SIf.In.bolPinDetected.intern = FALSE) AND (bolRE_PinDetected = TRUE) THEN
			bolRE_PinDetected := FALSE;
		END_IF

		//----------------------------------------------------------------------
		// Set section engaged (hanger in section)
		//----------------------------------------------------------------------
		
		// Wait for positive edge of the hanger sensor
		IF (SIf.In.bolHangerDetected.intern = TRUE) AND (bolRE_HangerDetected = FALSE) THEN
			bolRE_HangerDetected := TRUE;
				
			// Loop over section buffer to mark buffer element with 3 = section engaged (hanger in section detected by hanger sensor)
			FOR intSec := 0 TO Const_MTR.cusiSectionBuffer_SIZE-1 DO		
				
				// Prio 1: Normal sequence.
				IF (SIf.Par.dinHangerSensorPosition_um < a_stSectionBuffer[intSec].dinSecStartPos) AND  
					(SIf.Par.dinHangerSensorPosition_um > (a_stSectionBuffer[intSec].dinSecEndPos - SIf.Par.dinPinLenght_um)) THEN	
						// Mark the buffer element as engaged (hanger in section detected by hanger sensor)
						a_stSectionBuffer[intSec].enmState:= E_Typ_MTR_SECTION_STATE.EngagedByDetecSensor;
					EXIT;
				
				// Prio 2: If range is not accurately recognized mark buffer element X and X +1.
				ELSIF (SIf.Par.dinHangerSensorPosition_um < a_stSectionBuffer[intSec].dinSecEndPos) AND  
					(SIf.Par.dinHangerSensorPosition_um > a_stSectionBuffer[intSec+1].dinSecStartPos) THEN	
						// Mark the buffer element as engaged (hanger in section detected by hanger sensor)
						a_stSectionBuffer[intSec].enmState:= E_Typ_MTR_SECTION_STATE.EngagedByDetecSensor;
						a_stSectionBuffer[intSec+1].enmState:= E_Typ_MTR_SECTION_STATE.EngagedByDetecSensor;
					EXIT;
				END_IF		
					
			END_FOR	
				
		ELSIF (SIf.In.bolHangerDetected.intern = FALSE) AND (bolRE_HangerDetected = TRUE) THEN
			bolRE_HangerDetected := FALSE;
		END_IF	
		
		//----------------------------------------------------------------------
		// Buffer tracking 
		//----------------------------------------------------------------------
		
		// Move all buffer elements 1 down if section is driven out at the last line!		
		IF  (a_stSectionBuffer[0].enmState = E_Typ_MTR_SECTION_STATE.HangerReleased) OR (a_stSectionBuffer[0].dinSecEndPos > (dinPositionOfLastLine_um + SIf.Par.dinSectionLenght_um))THEN
			// Loop every buffer element 1 Down
			FOR intSec := 0 TO Const_MTR.cusiSectionBuffer_SIZE-1 DO			
				a_stSectionBuffer[intSec].dinSecStartPos := a_stSectionBuffer[intSec+1].dinSecStartPos;
				a_stSectionBuffer[intSec].dinSecEndPos := a_stSectionBuffer[intSec+1].dinSecEndPos;
				a_stSectionBuffer[intSec].dinTrigStartPos := a_stSectionBuffer[intSec+1].dinTrigStartPos;
				a_stSectionBuffer[intSec].dinTrigEndPos := a_stSectionBuffer[intSec+1].dinTrigEndPos;		
				a_stSectionBuffer[intSec].usiReservedForLine:= a_stSectionBuffer[intSec+1].usiReservedForLine;			
				a_stSectionBuffer[intSec].enmState := a_stSectionBuffer[intSec+1].enmState;
			END_FOR		
			a_stSectionBuffer[intSec].dinSecStartPos := 0;
			a_stSectionBuffer[intSec].dinSecEndPos := 0;
			a_stSectionBuffer[intSec].dinTrigStartPos := 0;
			a_stSectionBuffer[intSec].dinTrigEndPos := 0;
			a_stSectionBuffer[intSec].usiReservedForLine := 0;
			a_stSectionBuffer[intSec].enmState := E_Typ_MTR_SECTION_STATE.Undefined;
		END_IF
	
		//----------------------------------------------------------------------
		// Increase section positions
		//----------------------------------------------------------------------
		
		// Increase section positions and reserve sections
		FOR intSec := 0 TO Const_MTR.cusiSectionBuffer_SIZE DO
			IF (a_stSectionBuffer[intSec].enmState = E_Typ_MTR_SECTION_STATE.StartPositionSet) THEN
				// Section start/end
				a_stSectionBuffer[intSec].dinSecStartPos:= a_stSectionBuffer[intSec].dinSecStartPos + dinDrivenWay_um;
				// Trigger start/end
				a_stSectionBuffer[intSec].dinTrigStartPos:= a_stSectionBuffer[intSec].dinSecStartPos - SIf.Par.dinTrigStartOffset_um;
				a_stSectionBuffer[intSec].dinTrigEndPos:= a_stSectionBuffer[intSec].dinSecStartPos - SIf.Par.dinTrigEndOffset_um;	
				
			ELSIF (a_stSectionBuffer[intSec].enmState >= E_Typ_MTR_SECTION_STATE.EndPositionSet) THEN
				// Section start/end
				a_stSectionBuffer[intSec].dinSecStartPos:= a_stSectionBuffer[intSec].dinSecStartPos + dinDrivenWay_um;
				a_stSectionBuffer[intSec].dinSecEndPos:= a_stSectionBuffer[intSec].dinSecEndPos + dinDrivenWay_um;
				// Trigger start/end
				a_stSectionBuffer[intSec].dinTrigStartPos:= a_stSectionBuffer[intSec].dinSecStartPos - SIf.Par.dinTrigStartOffset_um;
				a_stSectionBuffer[intSec].dinTrigEndPos:= a_stSectionBuffer[intSec].dinSecStartPos - SIf.Par.dinTrigEndOffset_um;
			END_IF
		END_FOR

		//-------------------------------------------------------------------------------------
		// Handle reservation for a section, also clear reservations if no hanger exist 
		//-------------------------------------------------------------------------------------
		
		FOR intSec := 0 TO Const_MTR.cusiSectionBuffer_SIZE DO

			// Note: If the section end passed the position of the hanger detection sensor, the section is not engaged and the section start pos. is before position of the first line, 
			// then the section can reserved for a line.
			IF (a_stSectionBuffer[intSec].enmState = E_Typ_MTR_SECTION_STATE.EndPositionSet) AND 
			   (a_stSectionBuffer[intSec].dinSecEndPos > SIf.Par.dinHangerSensorPosition_um) THEN 
			  // (a_stSectionBuffer[intSec].dinSecStartPos < a_pLineChildSIF[0]^.Par.dinPositionOfSlide_um) THEN   	// ToDO: DSC, test
			
	
				bolExit:= FALSE;	
				WHILE (NOT bolExit) DO						
					IF (intLine <= (usiNumOfLines-1)) THEN			
			
						// Check if hanger exist on line
						// .............................
						IF (a_pLineChildSIF[intLine]^.Cur.bolHangerDetected) THEN
										
							IF (a_stSectionBuffer[intSec].dinSecStartPos < a_pLineChildSIF[intLine]^.Par.dinPositionOfSlide_um) THEN	// ToDO: DSC, test
								// Reserve a section for this line
								intLineNum:= intLine + 1;
								a_stSectionBuffer[intSec].usiReservedForLine:= INT_TO_USINT(intLineNum);
								a_stSectionBuffer[intSec].enmState:= E_Typ_MTR_SECTION_STATE.Reserved;
							END_IF
							
							// Set start index for next cycle
							IF (intLine < (usiNumOfLines-1)) THEN
								intLine:= intLine + 1;	
							ELSE
								intLine:= 0;
							END_IF
							// -> Exit
							bolExit:= TRUE;
							
						// No hanger exist (no further hanger)
						// ............................
						ELSE
							// Delete existing reservations for this line. Make new space for other lines. 
							FOR intDeleteRes := 0 TO Const_MTR.cusiSectionBuffer_SIZE DO
								// Check if a section is already reserved for this line
								IF ((a_stSectionBuffer[intDeleteRes].enmState = E_Typ_MTR_SECTION_STATE.Reserved) AND (a_stSectionBuffer[intDeleteRes].usiReservedForLine = INT_TO_USINT(intLine+1))) THEN
									// Delete reservation
									a_stSectionBuffer[intDeleteRes].usiReservedForLine:= 0;
									a_stSectionBuffer[intDeleteRes].enmState:= E_Typ_MTR_SECTION_STATE.EndPositionSet;			
								END_IF						
							END_FOR
						END_IF	
						// Inc. index to next line
						intLine:= intLine + 1;				
					ELSE
						// Start again at first line	
						intLine:= 0;
						bolExit:= TRUE;
					END_IF				
				END_WHILE		
								
			END_IF

		END_FOR

		// Check States for parent information
		THIS^.checkStateAllLines(cSTA_RUN);
		
		// State Change Condition
		IF (me.intCmd=cCMD_STOP) THEN
			me.StateMachine.intStateNext := cSTA_STOPBusy;
		END_IF
		
	END_IF

//--------------------------------------------------------------------------------------
// Exit action
	IF (me.StateMachine.intState<>me.StateMachine.intStateNext) THEN
		;
	END_IF
END_METHOD

METHOD PROTECTED sta_RUNBusy : BOOL
VAR
	ii: INT;
END_VAR
// state implemetation
//--------------------------------------------------------------------------------------
// Entry action
	IF (me.StateMachine.intState<>me.StateMachine.intStateLastCycle) THEN
		me.StateMachine.intStateLastCycle := me.StateMachine.intState;
		;
	END_IF

//--------------------------------------------------------------------------------------
// Cyclic action
	IF (me.StateMachine.intState=me.StateMachine.intStateLastCycle) THEN
			
		// Clear section buffer
		FOR ii := 0 TO Const_MTR.cusiSectionBuffer_SIZE DO
			a_stSectionBuffer[ii].dinSecStartPos := 0;
			a_stSectionBuffer[ii].dinSecEndPos := 0;
			a_stSectionBuffer[ii].dinTrigStartPos := 0;
			a_stSectionBuffer[ii].dinTrigEndPos := 0;
			a_stSectionBuffer[ii].enmState := E_Typ_MTR_SECTION_STATE.Undefined;
			a_stSectionBuffer[ii].usiReservedForLine:= 0;
		END_FOR
			
		// send command RUN to all existing line child controller.
		THIS^.CmdToAllLines(cCMD_RUN);
			
		// State Change Condition	
		IF (THIS^.checkStateAllLines(cSTA_RUN)) THEN
			me.StateMachine.intStateNext := cSTA_RUN;		
		END_IF

	END_IF

//--------------------------------------------------------------------------------------
// Exit action
	IF (me.StateMachine.intState<>me.StateMachine.intStateNext) THEN
		;
	END_IF
END_METHOD

METHOD PROTECTED sta_STOP : BOOL
// state implemetation
//--------------------------------------------------------------------------------------
// Entry action
	IF (me.StateMachine.intState<>me.StateMachine.intStateLastCycle) THEN
		me.StateMachine.intStateLastCycle := me.StateMachine.intState;
		;
	END_IF

//--------------------------------------------------------------------------------------
// Cyclic action
	IF (me.StateMachine.intState=me.StateMachine.intStateLastCycle) THEN

		// State Change Condition	
		IF (me.intCmd = cCMD_RUN) THEN 
			me.StateMachine.intStateNext := cSTA_RUNBusy;
		END_IF
	END_IF

//-------------------------------------------------------------------------------------
// Exit action
	IF (me.StateMachine.intState<>me.StateMachine.intStateNext) THEN
		;
	END_IF
END_METHOD

METHOD PROTECTED sta_STOPBusy : BOOL
// state implemetation
//--------------------------------------------------------------------------------------
// Entry action
	IF (me.StateMachine.intState<>me.StateMachine.intStateLastCycle) THEN
		me.StateMachine.intStateLastCycle := me.StateMachine.intState;
		
		// send command STOP to all existing line child controller.
		THIS^.CmdToAllLines(cCMD_STOP);

	END_IF

//--------------------------------------------------------------------------------------
// Cyclic action
	IF (me.StateMachine.intState=me.StateMachine.intStateLastCycle) THEN
			
		// State Change Condition
		// Check if all STOPPED
		IF (THIS^.checkStateAllLines(cSTA_STOP)) THEN
			me.StateMachine.intStateNext := cSTA_STOP;
		END_IF
	END_IF

//--------------------------------------------------------------------------------------
// Exit action
	IF (me.StateMachine.intState<>me.StateMachine.intStateNext) THEN
		;
	END_IF
END_METHOD

METHOD PROTECTED StateMachine : BOOL
SUPER^.StateMachine();

// main statemachine of base controller
CASE me.StateMachine.intState OF
    cSTA_STOPBusy: 
        THIS^.sta_STOPBusy();
    cSTA_STOP: 
        THIS^.sta_STOP();
	cSTA_RUNBusy: 
        THIS^.sta_RUNBusy();
    cSTA_RUN: 
        THIS^.sta_RUN();				
END_CASE;
END_METHOD

END_FUNCTION_BLOCK

// POUs/Controller/Lvl2/MER (Merger Standard)/FB_MER
FUNCTION_BLOCK FB_MER EXTENDS FB_CtrlBase IMPLEMENTS IBuffer
VAR_INPUT
	/// Sensors for jam detection
	In_a_bolJamSensor: ARRAY[1..cMAX_JAM_SENSORS] OF BOOL;
END_VAR
VAR
	/// Specific interface struct for public access
	SIf: T_Ctrl_SIf_MER;
	/// List of pointers to Childs
	a_pLineChildCtrl: ARRAY[0..Base_Const.cMaxNrOfChilds] OF POINTER TO FB_SLB;
	/// List of childs common interface
	a_pLineChildCIF: ARRAY[0..Base_Const.cMaxNrOfChilds] OF POINTER TO T_Ctrl_CIf;
	/// List of childs specific interface for additional parameters or cur
	a_pLineChildSIF: ARRAY[0..Base_Const.cMaxNrOfChilds] OF POINTER TO T_Ctrl_SIf_SLB;
	/// Function specific variables
	usiNumOfLines: USINT;
	usiNumOfValidPointerToLine: USINT;
	bolHangerExist: BOOL;
	bolGoToRun: BOOL;
	dinPassedTotalLineXOld: DINT;
	/// Used for counting passed hangers if "E_Typ_MER_MODE.MergeOverSetpoint" is selected.
	dinNumOfPassedHangers: DINT;
	/// Used for time measurement if "E_Typ_MER_MODE.MergeOverTime" is selected.
	udiMergingTime: UDINT;
	usiLineNumToReleaseAll: USINT;
	usiIndexToRelease: USINT;
	bolReleaseHanger: BOOL;
	/// Shadow copy of In_a_bolJamSensor[]
	a_bolJamSensorOnce: ARRAY[1..cMAX_JAM_SENSORS] OF BOOL;
	/// Start time of jam sensor is true
	a_udiTimeJamDetection: ARRAY[1..cMAX_JAM_SENSORS] OF UDINT;
	/// Jam release delay timer
	udiJamReleaseDelayTime_ms: UDINT;
	/// Jam at merger output detected 
	bolJamDetected: BOOL;
	/// Loop variable
	intI: INT;
END_VAR
VAR CONSTANT
	/// sub States
	cSTA_SUB_INITIALIZED: INT := 500;
	cSTA_SUB_WAIT_FOR_CMD: INT := 502;
	cSTA_SUB_CHECK_HANGER_EXIST: INT := 504;
	cSTA_SUB_SEND_RELEASE: INT := 506;
	cSTA_SUB_SEND_RELEASE_ALL: INT := 508;
	cSTA_SUB_SEND_STOP: INT := 510;
	cSTA_SUB_WAIT_JOB_DONE: INT := 512;
	cSTA_SUB_CHECK_MERGE_CON: INT := 514;
	cSTA_SUB_WAIT_LINE_FREE: INT := 516;
	cSTA_SUB_END: INT := 518;
END_VAR

(*__________________________________________________________________________________________________
¦	
¦	Vistaprint Schweiz GmbH
¦	CH - 8401 Winterthur
¦
¦	www.vistaprint.ch - info@vistaprint.ch
¦___________________________________________________________________________________________________

Function desription:
The controller automatically merge hangers from different lines dependent time or distribution of the number of hangers.
Lines are always from controller type slide buffer FB_SLB.

History:
Version		Date			Author		Comment
---------------------------------------------------------------------------------------------------
0.00.1		05.09.2013		AVME/DSC	Start history. 
0.00.2		09.09.2013		AVME/DSC 	Integration of all merger basic functionalities. Test on simulator.
										Controller can work in 2 different main modes:
										-> "automatic", controller automatically merge hangers from different lines dependent E_Typ_MER_AUTO_MODE
										-> "on command", in case if merger work as charge controller. Release line X dependent from parent command.
0.00.3		19.09.2013		AVME/PRE	Implement new Base Concept
0.00.4		01.10.2013		AVME/DSC	Sub state machine general handling deleted. Not used anymore. Handled in Base Class.										
0.00.5		03.10.2013		AVME/PRE	Integrate new function insert Belt		
0.00.6		03.10.2013		AVME/PRE	Insert new sub state LOCK_SECTION.	
0.00.7		15.10.2013		AVME/DSC	Complete redesign of the merger "MergeIntoTrp" mode.
0.00.8		30.10.2013		AVME/DSC	Modifications for "MergeIntoTrp" mode during test at the tool. Good merging possible with drive speed = 0. (slow speed)
										Merging with higher speed not possible!				
0.00.9		08.11.2013		AVME/MRU	Stop merger if outfeed sensor detect a jam (Bugzilla Nr. 8)
0.00.10		03.12.2013		AVME/MRU	Add MaxCapacity / NumOfHangers properties
0.00.11		09.12.2013		AVME/DSC	Modification in method "checkStateAllLines".
										Special condition: In case if the child is in state ERROR and STOP is requested. Set child as checked.
										Parent controller need state STOP that automatic stop sequence can work for all other childs.
0.00.12		13.01.2014		AVME/MRU	Bugzilla ID 03: BufferFull for LineControl added
0.00.13		22.01.2014		AVME/MRU	udiJamReleaseDelayTime_ms added; Timing "Check jam detection" reworked
0.00.14		30.04.2014		AVME/DSC    Deleted complete handling for mode "MergeIntoTrp" and implemented function into new controller FB_MTR.									
__________________________________________________________________________________________________*)


IF ((me.bolActivate) AND (THIS^.checkChildValid())) THEN // cyclic call enabled
	IF (CIf.Info.bolInitDone=FALSE) THEN // first cycle -> init
		CtrlInit();
		CIf.Info.bolInitDone := TRUE;
	ELSE
		CycleStartDuty();
	
		Always();
		
		StateMachine();
		
		CycleEndDuty();
	END_IF
END_IF;

METHOD AddLine
VAR_INPUT
	p_Line: POINTER TO FB_SLB;
END_VAR

// Method add the pointer address of the line child controller to the array list.
IF (usiNumOfLines <= (Base_Const.cMaxNrOfChilds-1)) THEN
	// Add line child controller to list
	a_pLineChildCtrl[usiNumOfLines] := p_Line;
	// Inc. number of lines
	usiNumOfLines:= usiNumOfLines+1;
	// Check if the pointer is valid
	IF (p_Line<>0) THEN
		usiNumOfValidPointerToLine:= usiNumOfValidPointerToLine+1;
	END_IF
END_IF
END_METHOD

METHOD PROTECTED Always : BOOL
VAR
	/// Looping variable
	intSec: INT;
END_VAR
IF (me.bolChangeBackToAUTO=TRUE) THEN // switch mode to automatic switch off controller
	//me.StateMachine.intStateNext := cSTA_OFFBusy;
	//me.bolChangeBackToAUTO := FALSE; // for cylinder no change to off when switch to automatic!!
END_IF

SUPER^.Always();

// ----------------------------------------------------------------------------------
// cyclic actions outside of statemachine
IF (me.StateMachine.intState<>cSTA_SINGLE_ANSWER) THEN
	
	//-------------------------------------------------
	// Provide current values for the parent
	//-------------------------------------------------	
	
	// Number of lines to merge, depends on how many times the method "AddLine" was called at init
	SIf.Cur.usiNumOfLinesToMerge:= usiNumOfLines;
	// Actual Item Count of this controller -> based on all lines
	SIf.Cur.dinCurrentItemCount:= THIS^.CalcSumOfItems();
	// Max. buffer capacity -> based on all lines
	SIf.Cur.dinMaxCapacity:= THIS^.CalcMaxCapacity();	
	
END_IF

// ----------------------------------------------------------------------------------
// Always change actions in Base Library
// ----------------------------------------------------------------------------------
// overrule error always from base -> no EOFF State!! in EOFF go to OFF
IF (me.StateMachine.intStateNext = cSTA_EOFFBusy) THEN
	IF (me.StateMachine.intState=cSTA_OFF) THEN
		me.StateMachine.intStateNext := cSTA_OFF;
	ELSE // stay in OFF
		me.StateMachine.intStateNext := cSTA_OFFBusy;
	END_IF
END_IF

// Conditions Always
IF (((me.Alarm.eActivAlmClass=E_AlmClass.EOFF) OR (me.Alarm.eActivAlmClass=E_AlmClass.OFF) OR (me.intCmd=cCMD_OFF))
		 AND (me.StateMachine.intState<>cSTA_ERROR) AND (me.StateMachine.intState<>cSTA_ERRORQuit) AND
		(me.StateMachine.intState<>cSTA_OFF) AND (me.StateMachine.intState<>cSTA_OFFBusy)) THEN
	// alarm evt EOFF, OFF or cmd off
	me.StateMachine.intStateNext := cSTA_OFFBusy;
END_IF
END_METHOD

PROPERTY BufferFull : BOOL
GET
BufferFull:= False;
END_GET
END_PROPERTY

METHOD PROTECTED CalcMaxCapacity : DINT
VAR
	ii: INT;
	dinSumMaxCapacity: DINT;
END_VAR
// Method calculate the sum of max. capacities from all lines and return the result.

//Init
CalcMaxCapacity:= 0;
dinSumMaxCapacity:= 0;

// Loop over all childs
FOR ii:=0 TO usiNumOfLines-1 BY 1 DO
	// Build sum of all lines		
	dinSumMaxCapacity:= dinSumMaxCapacity + a_pLineChildSIF[ii]^.Cur.dinMaxCapacity; 	
END_FOR

// Return result
CalcMaxCapacity:= dinSumMaxCapacity;
END_METHOD

METHOD PROTECTED CalcSumOfItems : DINT
VAR
	ii: INT;
	dinSumOfItems: DINT;
END_VAR
// Method calculate the sum of hangers from all lines and return the result.

//Init
CalcSumOfItems:= 0;
dinSumOfItems:= 0;

// Loop over all childs
FOR ii:=0 TO usiNumOfLines-1 BY 1 DO
	// Build sum of all zones		
	dinSumOfItems:= dinSumOfItems + a_pLineChildSIF[ii]^.Cur.dinNumOfHangersInBuffer; 	
END_FOR

// Return result
CalcSumOfItems:= dinSumOfItems;
END_METHOD

METHOD checkChildAlmClass : BOOL
//------------------------------------------------------------------------------------------------------
// check child alarm classes
// set me alarm class active if at least one child has an EOFF
IF CheckAllChildAlmClass(E_AlmClass.EOFF) THEN
	CIf.Job.eMe_ActivAlmClass := E_AlmClass.EOFF;
	me.Alarm.bolfp := TRUE;
ELSIF CheckAllChildAlmClass(E_AlmClass.OFF) THEN
	CIf.Job.eMe_ActivAlmClass := E_AlmClass.OFF;
	me.Alarm.bolfp := TRUE;
ELSIF CheckAllChildAlmClass(E_AlmClass.STOP) THEN  // FB_MER needs alarm class STOP
	CIf.Job.eMe_ActivAlmClass := E_AlmClass.STOP;
	me.Alarm.bolfp := TRUE;
ELSE
	IF (me.Alarm.bolfp) THEN
		CIf.Job.eMe_ActivAlmClass := E_AlmClass.NONE; // no reset necessary
		me.Alarm.bolfp := FALSE;
	END_IF
END_IF

//------------------------------------------------------------------------------------------------------
// set alarm class parent of childs
//------------------------------------------------------------------------------------------------------
// set alarm class parent of childs in the case of a parent EOFF or me=OFF or EOFF
IF (CIf.Job.eParent_ActivAlmClass=E_AlmClass.EOFF) THEN
	SetAllChildAlmClass(CIf.Job.eParent_ActivAlmClass);
ELSIF(CIf.Job.eMe_ActivAlmClass=E_AlmClass.EOFF) OR (CIf.Job.eMe_ActivAlmClass=E_AlmClass.OFF) THEN
	SetAllChildAlmClass(CIf.Job.eMe_ActivAlmClass);
ELSE
	// no important alarm for child active
	SetAllChildAlmClass(E_AlmClass.NONE);
END_IF
END_METHOD

METHOD PROTECTED checkChildValid : BOOL
IF (usiNumOfLines = usiNumOfValidPointerToLine) THEN
	checkChildValid:= TRUE;
ELSE
	checkChildValid:= FALSE;
	// Invalid child pointer
	IF (usiNumOfLines <> usiNumOfValidPointerToLine) THEN
		// SIf.Alm[1].strText := 'Invalid child pointer'; 
		pfbAlarmCtrl^.setAlarm(CIf.Info.intCtrlId,1,0,ADR(SIf.Alm),E_AlmState.RST,CIf.Job.eMe_ActivAlmClass);	
	END_IF
END_IF
END_METHOD

METHOD PROTECTED checkStateAllLines : BOOL
VAR_INPUT
	cSTA: INT;
END_VAR
VAR
	ii: INT;
	usiNumOfCheckedChilds: USINT;
END_VAR
// Method check input state of all lines

//Init
checkStateAllLines:= FALSE;
usiNumOfCheckedChilds:= 0;

// Loop over all childs
FOR ii:=0 TO usiNumOfLines-1 BY 1 DO
	// Check state	
	// Special condition: In case if the child is in state ERROR and STOP is requested. Set child as checked.
	// Parent controller need state STOP that automatic stop sequence can work for all other childs.
	IF (a_pLineChildCIF[ii]^.Job.intState = cSTA) OR ((a_pLineChildCIF[ii]^.Job.intState = cSTA_ERROR) AND (cSTA = cSTA_STOP)) THEN
		usiNumOfCheckedChilds:= usiNumOfCheckedChilds+1;
		SIf.Cur.a_bolChildReady[ii] := TRUE;
	ELSE
		SIf.Cur.a_bolChildReady[ii] := FALSE;		
	END_IF

END_FOR

// All states equal the input state
IF (usiNumOfCheckedChilds = usiNumOfLines) THEN
	checkStateAllLines:= TRUE;
END_IF
END_METHOD

METHOD PROTECTED CmdToAllLines
VAR_INPUT
	cCMD: INT;
END_VAR
VAR
	ii: INT;
END_VAR
// Method send input command to all existing line child controller.
FOR ii:=0 TO usiNumOfLines-1 BY 1 DO	
	a_pLineChildCIF[ii]^.Job.intACmd:= cCMD;
END_FOR
END_METHOD

METHOD PROTECTED CtrlInit : BOOL
VAR
	ii: INT;
END_VAR
SUPER^.CtrlInit();

//----------------------------------------------------------------------
// Initialize all lines
//----------------------------------------------------------------------

// Method initialize all line child controller.
FOR ii:=0 TO usiNumOfLines-1 BY 1 DO	
	a_pLineChildCIF[ii] := THIS^.AddChild(a_pLineChildCtrl[ii]^);
	a_pLineChildSIF[ii] := a_pLineChildCtrl[ii]^.getCtrlSIf();
END_FOR
END_METHOD

METHOD FB_init : BOOL
VAR_INPUT
	///if TRUE, the retain variables are initialized (warm start / cold start)
	bInitRetains: BOOL;
	///if TRUE, the instance afterwards gets moved into the copy code (online change)
	bInCopyCode: BOOL;
END_VAR
VAR
	ii: UINT;
END_VAR
//------------------------------------------------------------------------------------------------------------------------
// to manually change in new FUB implementation!!!
// define valid commands for this controller
FOR ii:= 0 TO (SIZEOF(CIf.Job.aCmdList)/SIZEOF(CIf.Job.aCmdList[0])-1) BY 1 DO
	IF (CIf.Job.aCmdList[ii].intCmd=cCMD_INITIALIZED) THEN
		// found first empty array element
		EXIT;
	END_IF
END_FOR

CIf.Job.aCmdList[ii].intCmd := cCMD_STOP;
CIf.Job.aCmdList[ii].strName := 'Stop'; 
CIf.Job.aCmdList[ii].bolAvailable := TRUE;
ii := ii +1;
CIf.Job.aCmdList[ii].intCmd := cCMD_RUN;
CIf.Job.aCmdList[ii].strName := 'Run';
CIf.Job.aCmdList[ii].bolAvailable := TRUE;

// set name of class/typ
CIf.Info.strType := 'FB_MER'; 

// set alarm class
SIf.Alm[1].eAlmClass := E_AlmClass.STOP;
SIf.Alm[1].strText := 'Invalid child pointer';
SIf.Alm[2].eAlmClass := E_AlmClass.INFO;
SIf.Alm[2].strText := 'Invalid line number. Line not exist';
SIf.Alm[3].eAlmClass := E_AlmClass.INFO;
SIf.Alm[3].strText := 'Merger waits for jam sensor free'; 


//*******************************************************************************
// initial values
//*******************************************************************************

// software configuration
CIf.SwCfg.bolExist := TRUE;
CIf.SwCfg.bolSimulation := FALSE;

// configuration
SIf.Cfg.usiMergeMainMode:= E_Typ_MER_MODE.Automatic;
SIf.Cfg.usiCountJamSensors:= 0;

// parameter
SIf.Par.udi_jamTimeout_ms:= 500;
// Default parameter for the lines are set in method InitLines
END_METHOD

METHOD PROTECTED getCmdState : STRING
VAR_INPUT
	intCmdState: INT;
	bolState: BOOL;
END_VAR
getCmdState := SUPER^.getCmdState(intCmdState:=intCmdState,bolState:=bolState); // get global/base defined cmds/states
IF (getCmdState='') THEN // global not defined get local
	// get string cmd/state string information in runtime
	IF (bolState=FALSE) THEN
		// cmd's
		CASE intCmdState OF
		END_CASE;
	ELSE
	
	// states
		CASE intCmdState OF	
			// SUB States
			cSTA_SUB_INITIALIZED:
				getCmdState := 'cSTA_SUB_INITIALIZED';			
			cSTA_SUB_WAIT_FOR_CMD:
				getCmdState := 'cSTA_SUB_WAIT_FOR_CMD';					
			cSTA_SUB_CHECK_HANGER_EXIST:
				getCmdState := 'cSTA_SUB_CHECK_HANGER_EXIST';
			cSTA_SUB_SEND_RELEASE:
				getCmdState := 'cSTA_SUB_SEND_RELEASE';
			cSTA_SUB_SEND_RELEASE_ALL:
				getCmdState := 'cSTA_SUB_SEND_RELEASE_ALL';	
			cSTA_SUB_SEND_STOP:
				getCmdState := 'cSTA_SUB_SEND_STOP';		
			cSTA_SUB_WAIT_JOB_DONE:
				getCmdState := 'cSTA_SUB_WAIT_JOB_DONE';
			cSTA_SUB_CHECK_MERGE_CON:
				getCmdState := 'cSTA_SUB_CHECK_MERGE_CON';
			cSTA_SUB_WAIT_LINE_FREE:
				getCmdState := 'cSTA_SUB_WAIT_LINE_FREE';	
			cSTA_SUB_END:
				getCmdState := 'cSTA_SUB_END';	
		END_CASE;
	END_IF
END_IF
END_METHOD

METHOD getCtrlSIf : POINTER TO T_Ctrl_SIf_MER
getCtrlSIf := ADR(SIf);
END_METHOD

METHOD PROTECTED IoInBridge : BOOL
// digitale and analoge inputs read from hardware or forcing
// Read sensors for waiting if a jam is detected
FOR intI := 1 TO SIf.Cfg.usiCountJamSensors DO
	SIf.In.a_bolJamSensor[intI].map := THIS^.In_a_bolJamSensor[intI];
	IF (CIf.SwCfg.bolSimulation = FALSE) THEN
		getInBol(CIf.Job.bolIoForce,ADR(SIf.In.a_bolJamSensor[intI]));
	END_IF
END_FOR

IF (CIf.SwCfg.bolSimulation = FALSE) THEN
	//ctrl.In.bol_PosSwitchBasicDefTyp.intern := getInBol(ctrl.ifc.Job.bol_Force ,ADR(ctrl.In.bol_PosSwitchBasicDefTyp);
ELSE
	//simulation of global IO
END_IF
END_METHOD

METHOD PROTECTED IoOutBridge : BOOL
// digitale and analoge inputs read from hardware or forcing

// ... no physical outputs

IF (CIf.SwCfg.bolSimulation = FALSE) THEN
	// check interlocks to prevent damages
	IF (CIf.Job.bolIlkOverwrite=FALSE) THEN
		;
	END_IF
END_IF
END_METHOD

PROPERTY MaxCapacity : DINT
GET
MaxCapacity:= SIf.Cur.dinMaxCapacity;
END_GET
END_PROPERTY

PROPERTY NumOfHangers : DINT
GET
NumOfHangers:= SIf.Cur.dinCurrentItemCount;
END_GET
END_PROPERTY

METHOD PROTECTED sta_OFF : BOOL
// state implemetation
//--------------------------------------------------------------------------------------
// Entry action
	IF (me.StateMachine.intState<>me.StateMachine.intStateLastCycle) THEN
		me.StateMachine.intStateLastCycle := me.StateMachine.intState;
		;		
	END_IF

//--------------------------------------------------------------------------------------
// Cyclic action
	IF (me.StateMachine.intState=me.StateMachine.intStateLastCycle) THEN
		
		// Reset total counter
		SIf.Cur.dinNumOfMergedHangersTotal:= 0;
		
		// State Change Condition
		IF (me.Alarm.eActivAlmClass<>E_AlmClass.EOFF) AND (me.Alarm.eActivAlmClass<>E_AlmClass.OFF) THEN
			IF (me.intCmd=cCMD_STOP) THEN
				me.StateMachine.intStateNext := cSTA_STOPBusy;
			ELSIF (me.intCmd=cCMD_RUN) THEN 
				me.StateMachine.intStateNext := cSTA_RUNBusy;
			END_IF
		END_IF
	END_IF

//--------------------------------------------------------------------------------------
// Exit action
	IF (me.StateMachine.intState<>me.StateMachine.intStateNext) THEN
		;
	END_IF
END_METHOD

METHOD PROTECTED sta_RUN : BOOL
// state implemetation
//--------------------------------------------------------------------------------------
// Entry action
	IF (me.StateMachine.intState<>me.StateMachine.intStateLastCycle) THEN
		me.StateMachine.intStateLastCycle := me.StateMachine.intState;	
		;
	END_IF

//--------------------------------------------------------------------------------------
// Cyclic action
	IF (me.StateMachine.intState=me.StateMachine.intStateLastCycle) THEN
			
	
		// Check States for parent information
		THIS^.checkStateAllLines(cSTA_RUN);

		// Check jam detection
		IF (udiJamReleaseDelayTime_ms > SIf.Par.udi_jamTimeout_ms) THEN
			bolJamDetected := FALSE;
		ELSE
			udiJamReleaseDelayTime_ms := udiJamReleaseDelayTime_ms + me.FUBInfo.udiSample_ms;
		END_IF
		
		FOR intI := 1 TO SIf.Cfg.usiCountJamSensors DO
			// Start jam timer
			IF ((SIf.In.a_bolJamSensor[intI].intern = TRUE) AND (a_bolJamSensorOnce[intI] = FALSE)) THEN
				a_bolJamSensorOnce[intI]:= TRUE;
				//a_udiTimeJamDetection[intI]:= me.StateMachine.udiTimeInState_ms;
				a_udiTimeJamDetection[intI]:= 0;
			// Stop jam timer
			ELSIF ((SIf.In.a_bolJamSensor[intI].intern = FALSE) AND (a_bolJamSensorOnce[intI] = TRUE)) THEN
				a_bolJamSensorOnce[intI]:= FALSE;
			// Set flag if neccessary
			ELSIF ((SIf.In.a_bolJamSensor[intI].intern = TRUE) AND (a_bolJamSensorOnce[intI] = TRUE)) THEN
				//IF (me.StateMachine.udiTimeInState_ms > a_udiTimeJamDetection[intI] + SIf.Par.udi_jamTimeout_ms) THEN
				IF (a_udiTimeJamDetection[intI] > SIf.Par.udi_jamTimeout_ms) THEN
					bolJamDetected := TRUE;
					udiJamReleaseDelayTime_ms := 0;
				END_IF
			END_IF
			a_udiTimeJamDetection[intI]:= a_udiTimeJamDetection[intI]+ me.FUBInfo.udiSample_ms;
		END_FOR
	
		//----------------------------------------------------------------------------------------
		// Substates for merging lines dependent time or distribution of the number of hangers
		//----------------------------------------------------------------------------------------
		CASE me.SubStateMachine.intState OF
	
			//-----------------------------------------------
			// INITIALIZE 					(MODE: All modes)
			//-----------------------------------------------
			cSTA_SUB_INITIALIZED:
			
				// Check configured main mode
				CASE SIf.Cfg.usiMergeMainMode OF	
				
					// Mode - Automatic
					E_Typ_MER_MODE.Automatic:		
						me.SubStateMachine.intStateNext := cSTA_SUB_CHECK_HANGER_EXIST;					
									
					// Mode - OnCommand	
					E_Typ_MER_MODE.OnCommand:		
						me.SubStateMachine.intStateNext := cSTA_SUB_WAIT_FOR_CMD;
														
				END_CASE
			
			//-----------------------------------------------
			// WAIT FOR COMMAND 			(MODE: OnCommand)
			//-----------------------------------------------	
			cSTA_SUB_WAIT_FOR_CMD:
			
				// Wait for command to release all
				IF (me.intCmd=SLB_CmdState.cCMD_RELEASE_ALL) THEN
					// Check about valid line number
					IF ((SIf.Par.usiLineNumToReleaseAll = 0) OR (SIf.Par.usiLineNumToReleaseAll > usiNumOfLines)) THEN
						// Invalid line	
						// SIf.Alm[2].strText := 'Invalid line number. Line not exist'; 
						pfbAlarmCtrl^.setAlarm(CIf.Info.intCtrlId,2,0,ADR(SIf.Alm),E_AlmState.RST,CIf.Job.eMe_ActivAlmClass);		
					ELSE
						// Valid line	
						usiLineNumToReleaseAll:= SIf.Par.usiLineNumToReleaseAll-1;
						me.SubStateMachine.intStateNext := cSTA_SUB_SEND_RELEASE_ALL;
					END_IF
						
				END_IF
				
			//-----------------------------------------------
			// CHECK HANGER EXIST 			(MODE: Automatic)     
			//-----------------------------------------------
			cSTA_SUB_CHECK_HANGER_EXIST:
				// Entry action
				IF (me.SubStateMachine.intState<>me.SubStateMachine.intStateLastCycle) THEN
					me.SubStateMachine.intStateLastCycle := me.SubStateMachine.intState;							
					;						
				END_IF
				
				// Init
				bolReleaseHanger:= FALSE;
					
				// Check hanger exists on line
				IF (a_pLineChildSIF[usiIndexToRelease]^.Cur.bolHangerDetected=TRUE) THEN
					bolReleaseHanger:= TRUE;					
				ELSE		
					// No hanger on this line, check next
					IF (usiIndexToRelease < (usiNumOfLines-1)) THEN
						// Inc. index to next line
						usiIndexToRelease:= usiIndexToRelease + 1;	
					ELSE
						usiIndexToRelease:= 0;
					END_IF
				END_IF			
	
				// State Change Condition
				IF (bolReleaseHanger=TRUE) THEN
					me.SubStateMachine.intStateNext := cSTA_SUB_SEND_RELEASE;
					// Reset counter and timer
					dinNumOfPassedHangers:=0;
					udiMergingTime:=0;
				END_IF
					
			//-----------------------------------------------
			// SEND RELEASE					(MODE: Automatic)
			//-----------------------------------------------
			cSTA_SUB_SEND_RELEASE:		
	
				// Send release command to line X (trigger command)
				a_pLineChildCIF[usiIndexToRelease]^.Job.intACmd:= STB_CmdState.cCMD_RELEASE;				
				
				// State Change Condition
				IF(TRUE)THEN
					me.SubStateMachine.intStateNext := cSTA_SUB_WAIT_JOB_DONE;					
				END_IF	
						
			//-----------------------------------------------
			// SEND RELEASE	ALL				(MODE: OnCommand)
			//-----------------------------------------------
			cSTA_SUB_SEND_RELEASE_ALL:
			
				// Send release all command to line X
				a_pLineChildCIF[usiLineNumToReleaseAll]^.Job.intACmd:= STB_CmdState.cCMD_RELEASE_ALL;				
				
				// State Change Condition
				IF(TRUE)THEN
					me.SubStateMachine.intStateNext := cSTA_SUB_WAIT_JOB_DONE;					
				END_IF		
					
			//-----------------------------------------------
			// WAIT JOB DONE				(MODE: All modes)
			//-----------------------------------------------
			cSTA_SUB_WAIT_JOB_DONE:
		
				// Check configured main mode
				CASE SIf.Cfg.usiMergeMainMode OF	
				
					// Mode - Automatic
					E_Typ_MER_MODE.Automatic:
						// State Change Condition
						// Wait until job done
						IF(a_pLineChildCIF[usiIndexToRelease]^.Job.intACmd = cSTA_DONE) THEN									
							me.SubStateMachine.intStateNext := cSTA_SUB_CHECK_MERGE_CON;																				
						END_IF	
									
					// Mode - OnCommand	
					E_Typ_MER_MODE.OnCommand:
						// State Change Condition
						// Wait until release all
						IF(a_pLineChildCIF[usiLineNumToReleaseAll]^.Job.intState = SLB_CmdState.cCMD_RELEASE_ALL)THEN				
							me.SubStateMachine.intStateNext := cSTA_SUB_SEND_STOP;																
						END_IF
						
				END_CASE
							
			//-----------------------------------------------
			// SEND STOP					(MODE: OnCommand)
			//-----------------------------------------------
			cSTA_SUB_SEND_STOP:
			
				// Send stop command to line X
				a_pLineChildCIF[usiLineNumToReleaseAll]^.Job.intACmd:=cCMD_RUN;				
				
				// State Change Condition
				IF(a_pLineChildCIF[usiLineNumToReleaseAll]^.Job.intState=cSTA_RUN)THEN
					me.SubStateMachine.intStateNext := cSTA_SUB_WAIT_LINE_FREE;					
				END_IF	
								
			//-----------------------------------------------
			// CHECK MERGE CONDITIONS		(MODE: Automatic)
			//-----------------------------------------------
			cSTA_SUB_CHECK_MERGE_CON:
				// Entry action
				IF (me.SubStateMachine.intState<>me.SubStateMachine.intStateLastCycle) THEN
					me.SubStateMachine.intStateLastCycle := me.SubStateMachine.intState;							
					;						
				END_IF
					
				// Count the passed hangers from current line X
				IF (a_pLineChildSIF[usiIndexToRelease]^.Cur.dinHangersPassedTotal <> dinPassedTotalLineXOld) THEN
					// Count passed hangers if "E_Typ_MER_AUTO_MODE.MergeOverSetpoint" is selected.				
					dinNumOfPassedHangers:= dinNumOfPassedHangers + a_pLineChildSIF[usiIndexToRelease]^.Cur.uinNumOfHangersPerPulseFirstZone;			
					// Calculate merged hangers total
					SIf.Cur.dinNumOfMergedHangersTotal:= SIf.Cur.dinNumOfMergedHangersTotal + a_pLineChildSIF[usiIndexToRelease]^.Cur.uinNumOfHangersPerPulseFirstZone;									
				END_IF
				dinPassedTotalLineXOld:= a_pLineChildSIF[usiIndexToRelease]^.Cur.dinHangersPassedTotal;
		
					
				// State Change Condition
				IF (a_pLineChildSIF[usiIndexToRelease]^.Cur.bolHangerDetected=FALSE) THEN	// No hanger exist
					me.SubStateMachine.intStateNext := cSTA_SUB_WAIT_LINE_FREE;				
				ELSIF ((SIf.Par.a_LinePar[usiIndexToRelease].usiMergeMode = E_Typ_MER_AUTO_MODE.MergeOverTime) AND (udiMergingTime >= SIf.Par.a_LinePar[usiIndexToRelease].udiMergingTime_ms)) THEN
					me.SubStateMachine.intStateNext := cSTA_SUB_WAIT_LINE_FREE;				
				ELSIF ((SIf.Par.a_LinePar[usiIndexToRelease].usiMergeMode = E_Typ_MER_AUTO_MODE.MergeOverSetpoint) AND (dinNumOfPassedHangers >= SIf.Par.a_LinePar[usiIndexToRelease].uinNumOfHangersToMerge)) THEN
					me.SubStateMachine.intStateNext := cSTA_SUB_WAIT_LINE_FREE;							
				ELSIF ((SIf.Par.a_LinePar[usiIndexToRelease].usiMergeMode = E_Typ_MER_AUTO_MODE.MergeOverTime) AND (udiMergingTime < SIf.Par.a_LinePar[usiIndexToRelease].udiMergingTime_ms)) THEN
					me.SubStateMachine.intStateNext := cSTA_SUB_SEND_RELEASE;					
				ELSIF ((SIf.Par.a_LinePar[usiIndexToRelease].usiMergeMode = E_Typ_MER_AUTO_MODE.MergeOverSetpoint) AND (dinNumOfPassedHangers < SIf.Par.a_LinePar[usiIndexToRelease].uinNumOfHangersToMerge)) THEN
					me.SubStateMachine.intStateNext := cSTA_SUB_SEND_RELEASE;	
				END_IF
	
			//-----------------------------------------------
			// WAIT UNTIL LINE IS FREE		(MODE: All modes)
			//-----------------------------------------------
			cSTA_SUB_WAIT_LINE_FREE:

				IF (bolJamDetected	= TRUE) THEN // Line is not free, jam detected
					// SIf.Alm[3].strText := 'Merger waits for jam sensor free';
					pfbAlarmCtrl^.setAlarm(CIf.Info.intCtrlId,3,0,ADR(SIf.Alm),E_AlmState.RST,CIf.Job.eMe_ActivAlmClass);				
				ELSE				
					// Check configured main mode
					CASE SIf.Cfg.usiMergeMainMode OF	
					
						// Mode - Automatic
						E_Typ_MER_MODE.Automatic:
							// State Change Condition
							IF (me.SubStateMachine.udiTimeInState_ms > SIf.Par.a_LinePar[usiIndexToRelease].udiWaitTimeLineFree_ms) THEN 
								IF(me.intCmd=cCMD_STOP)THEN
									// Go to end
									me.SubStateMachine.intStateNext := cSTA_SUB_END;
								ELSE
									// Merging cycle line X complete
									IF (usiIndexToRelease < (usiNumOfLines-1)) THEN						
										// Inc. index to next line
										usiIndexToRelease:= usiIndexToRelease + 1;	
									ELSE
										usiIndexToRelease:= 0;
									END_IF
									
									// Go on with automatic cycle
									me.SubStateMachine.intStateNext := cSTA_SUB_CHECK_HANGER_EXIST;					
								END_IF		
							END_IF
									
						// Mode - OnCommand	
						E_Typ_MER_MODE.OnCommand:
							// State Change Condition
							IF (me.SubStateMachine.udiTimeInState_ms > SIf.Par.a_LinePar[usiLineNumToReleaseAll].udiWaitTimeLineFree_ms) THEN												
								// Update merged hangers total -> After release all, use passed package 
								SIf.Cur.dinNumOfMergedHangersTotal:= SIf.Cur.dinNumOfMergedHangersTotal + a_pLineChildSIF[usiLineNumToReleaseAll]^.Cur.dinHangersPassedPackage;			
								
								IF(me.intCmd=cCMD_STOP)THEN
									// Go to end
									me.SubStateMachine.intStateNext := cSTA_SUB_END;
								ELSE
									//Set "Job done" for parent
									CIf.Job.intACmd:=cSTA_DONE;
									me.SubStateMachine.intStateNext := cSTA_SUB_WAIT_FOR_CMD;
								END_IF								
							END_IF
							
					END_CASE
				END_IF
			//-----------------------------------------------
			// END							(MODE: All modes)
			//-----------------------------------------------
			cSTA_SUB_END:
			     // ... do nothing
		
		END_CASE

		// Timer handling for merging time
		udiMergingTime:= udiMergingTime + me.FUBInfo.udiSample_ms;
			
		// State Change Condition
		IF ((me.intCmd=cCMD_STOP) AND ((me.SubStateMachine.intState=cSTA_SUB_END) OR (me.SubStateMachine.intState=cSTA_SUB_CHECK_HANGER_EXIST) OR (me.SubStateMachine.intState=cSTA_SUB_WAIT_FOR_CMD) OR (me.SubStateMachine.intState=cSTA_SUB_WAIT_LINE_FREE))) THEN
			me.StateMachine.intStateNext := cSTA_STOPBusy;
		END_IF
	END_IF

//--------------------------------------------------------------------------------------
// Exit action
	IF (me.StateMachine.intState<>me.StateMachine.intStateNext) THEN
		;
	END_IF
END_METHOD

METHOD PROTECTED sta_RUNBusy : BOOL
VAR
	ii: INT;
END_VAR
// state implemetation
//--------------------------------------------------------------------------------------
// Entry action
	IF (me.StateMachine.intState<>me.StateMachine.intStateLastCycle) THEN
		me.StateMachine.intStateLastCycle := me.StateMachine.intState;
	
		bolGoToRun:= FALSE;
		usiIndexToRelease:= 0;
		
		// Initialize sub state machine
		me.SubStateMachine.intState:= cSTA_SUB_INITIALIZED; 
		me.SubStateMachine.intStateNext:= cSTA_SUB_INITIALIZED;
		
	END_IF

//--------------------------------------------------------------------------------------
// Cyclic action
	IF (me.StateMachine.intState=me.StateMachine.intStateLastCycle) THEN
					
		// Check configured main mode
		CASE SIf.Cfg.usiMergeMainMode OF	
		
			// Mode - Automatic
			E_Typ_MER_MODE.Automatic:
			
				// send command RUN to all existing line child controller.
				THIS^.CmdToAllLines(cCMD_RUN);
				
				// State Change Condition
				// Check if all childs in "RUN", ready for release hanger 
				IF(THIS^.checkStateAllLines(cSTA_RUN))THEN
					bolGoToRun:= TRUE;			
				END_IF	
		
			// Mode - OnCommand	
			E_Typ_MER_MODE.OnCommand:
			
				// send command STOP to all existing line child controller.
				THIS^.CmdToAllLines(cCMD_RUN);
				
				// State Change Condition
				// Check if all childs stopped, ready for new command 
				IF(THIS^.checkStateAllLines(cSTA_RUN))THEN
					bolGoToRun:= TRUE;					
				END_IF	
			
		END_CASE

	
		// State Change Condition	
		IF (bolGoToRun=TRUE) THEN
			me.StateMachine.intStateNext := cSTA_RUN;		
		END_IF

	END_IF

//--------------------------------------------------------------------------------------
// Exit action
	IF (me.StateMachine.intState<>me.StateMachine.intStateNext) THEN
		;
	END_IF
END_METHOD

METHOD PROTECTED sta_STOP : BOOL
// state implemetation
//--------------------------------------------------------------------------------------
// Entry action
	IF (me.StateMachine.intState<>me.StateMachine.intStateLastCycle) THEN
		me.StateMachine.intStateLastCycle := me.StateMachine.intState;
		;
	END_IF

//--------------------------------------------------------------------------------------
// Cyclic action
	IF (me.StateMachine.intState=me.StateMachine.intStateLastCycle) THEN

		// State Change Condition	
		IF (me.intCmd = cCMD_RUN) THEN 
			me.StateMachine.intStateNext := cSTA_RUNBusy;
		END_IF
	END_IF

//-------------------------------------------------------------------------------------
// Exit action
	IF (me.StateMachine.intState<>me.StateMachine.intStateNext) THEN
		;
	END_IF
END_METHOD

METHOD PROTECTED sta_STOPBusy : BOOL
// state implemetation
//--------------------------------------------------------------------------------------
// Entry action
	IF (me.StateMachine.intState<>me.StateMachine.intStateLastCycle) THEN
		me.StateMachine.intStateLastCycle := me.StateMachine.intState;
		
		// send command STOP to all existing line child controller.
		THIS^.CmdToAllLines(cCMD_STOP);

	END_IF

//--------------------------------------------------------------------------------------
// Cyclic action
	IF (me.StateMachine.intState=me.StateMachine.intStateLastCycle) THEN
			
		// State Change Condition
		// Check if all STOPPED
		IF (THIS^.checkStateAllLines(cSTA_STOP)) THEN
			me.StateMachine.intStateNext := cSTA_STOP;
		END_IF
	END_IF

//--------------------------------------------------------------------------------------
// Exit action
	IF (me.StateMachine.intState<>me.StateMachine.intStateNext) THEN
		;
	END_IF
END_METHOD

METHOD PROTECTED StateMachine : BOOL
SUPER^.StateMachine();

// main statemachine of base controller
CASE me.StateMachine.intState OF
    cSTA_STOPBusy: 
        THIS^.sta_STOPBusy();
    cSTA_STOP: 
        THIS^.sta_STOP();
	cSTA_RUNBusy: 
        THIS^.sta_RUNBusy();
    cSTA_RUN: 
        THIS^.sta_RUN();				
END_CASE;
END_METHOD

END_FUNCTION_BLOCK

// POUs/Controller/Lvl1/SLB (Slide buffer)/FB_SLB
FUNCTION_BLOCK FB_SLB EXTENDS FB_CtrlBase IMPLEMENTS IBuffer
VAR
	/// Specific interface struct for public access
	SIf: T_Ctrl_SIf_SLB;
	/// List of pointers to Childs
	a_pBufferZoneChildCtrl: ARRAY[0..Base_Const.cMaxNrOfChilds] OF POINTER TO FB_STB;
	/// List of childs common interface
	a_pBufferZoneChildCIF: ARRAY[0..Base_Const.cMaxNrOfChilds] OF POINTER TO T_Ctrl_CIf;
	/// List of childs specific interface for additional parameters or cur
	a_pBufferZoneChildSIF: ARRAY[0..Base_Const.cMaxNrOfChilds] OF POINTER TO T_Ctrl_SIf_STB;
	/// Function specific variables
	usiNumOfBufferZones: USINT;
	usiNumOfValidPointerToZone: USINT;
	bolAllZonesEmpty: BOOL;
	dinPassedTotalZone1Old: DINT;
	/// Var. used for sub sequence refill
	intIndexRefill: INT;
	SubStateMachineRefill: INT;
	udiTimeInStateRefill_ms: UDINT;
	/// Var. used for simulation
	abolRESimRetract: ARRAY[0..Base_Const.cMaxNrOfChilds] OF BOOL;
END_VAR
VAR CONSTANT
	/// sub States
	cSTA_SUB_WAIT_FOR_CMD: INT := 500;
	cSTA_SUB_SEND_RELEASE: INT := 502;
	cSTA_SUB_SEND_STOP: INT := 504;
	cSTA_SUB_BREAK: INT := 506;
END_VAR

(*__________________________________________________________________________________________________
¦	
¦	Vistaprint Schweiz GmbH
¦	CH - 8401 Winterthur
¦
¦	www.vistaprint.ch - info@vistaprint.ch
¦___________________________________________________________________________________________________

Function desription:
The slide buffer controller handles the automatic refill and sequential emptying of different buffer zones. 
Buffer zones may consist of the following components: Separator, Double Stopper or Single Stopper.

History:
Version		Date			Author		Comment
---------------------------------------------------------------------------------------------------
0.00.1		02.09.2013		AVME/DSC	Start history. 
0.00.2		04.09.2013		AVME/DSC	Integration of all slide buffer basic functionalities. 
										Test on simulator.
0.00.3		06.09.2013		AVME/DSC    Renaming of method checkChildPointer to checkChildValid.
										Insert add. validation to check if the number of added childs is valid.
										Slide buffer controller can now also used with only one buffer.
0.00.4 		09.09.2013		AVME/DSC    Copied content from state "RUN_busy" to "RUN".  
										Insert new method for calculation of the max. capacity for all childs.
0.00.5		10.09.2013		AVME/PRE	Implement Simulation
										Correct counter if buffer empty only if hanger detection sensor
										Give released item to next Buffer
0.00.6		19.09.2013		AVME/PRE	Implement new Base Concept
0.00.7		28.10.2013		VP/RE		SLB is full is last zone is full. Otherwise it leads to overflow problems.
0.00.8 		04.11.2013		AVME/DSC    Modified ".cur" interface. Newly distinction is made ​​between: "bolInputBufferFull" and  "bolAllBuffersFull"
0.00.9		03.12.2013		AVME/MRU	Add MaxCapacity / NumOfHangers properties
0.00.10		09.12.2013		AVME/DSC	Modification in method "checkStateAllZones".
										Special condition: In case if the child is in state ERROR and STOP is requested. Set child as checked.
										Parent controller need state STOP that automatic stop sequence can work for all other childs.
0.00.11		10.01.2014		AVME/MRU	Bugzilla ID 55: Refill aloud, if dinNumOfHangersInBuffer < dinMaxCapacity (Without uinNumOfHangersPerPulse)
0.00.12		13.01.2014		AVME/MRU	Bugzilla ID 03: BufferFull for LineControl added
										
__________________________________________________________________________________________________*)


IF ((me.bolActivate) AND (THIS^.checkChildValid())) THEN // cyclic call enabled
	IF (CIf.Info.bolInitDone=FALSE) THEN // first cycle -> init
		CtrlInit();
		CIf.Info.bolInitDone := TRUE;
	ELSE
		CycleStartDuty();
	
		Always();
		
		StateMachine();
		
		CycleEndDuty();
	END_IF
END_IF;

METHOD AddBufferZone
VAR_INPUT
	p_BufferZone: POINTER TO FB_STB;
END_VAR

// Method add the pointer address of the buffer zone child controller to the array list.
IF (usiNumOfBufferZones <= (Base_Const.cMaxNrOfChilds-1)) THEN
	// Add buffer zone child controller to list
	a_pBufferZoneChildCtrl[usiNumOfBufferZones] := p_BufferZone;
	// Inc. number of buffer zones
	usiNumOfBufferZones:= usiNumOfBufferZones+1;
	// Check if the pointer is valid
	IF (p_BufferZone<>0) THEN
		usiNumOfValidPointerToZone:= usiNumOfValidPointerToZone+1;
	END_IF
END_IF
END_METHOD

METHOD PROTECTED Always : BOOL
IF (me.bolChangeBackToAUTO=TRUE) THEN // switch mode to automatic switch off controller
	//me.StateMachine.intStateNext := cSTA_OFFBusy;
	//me.bolChangeBackToAUTO := FALSE; // for cylinder no change to off when switch to automatic!!
END_IF

SUPER^.Always();

// ----------------------------------------------------------------------------------
// cyclic actions outside of statemachine
IF (me.StateMachine.intState<>cSTA_SINGLE_ANSWER) THEN
	
	//-------------------------------------------------
	// Provide current values for the parent
	//-------------------------------------------------	
	
	// Number of buffer zones, depends on how many times the method "AddBufferZone" was called at init
	SIf.Cur.usiNumOfBufferZones:= usiNumOfBufferZones;
	// Input buffer is full -> based on last zone full signal
	SIf.Cur.bolInputBufferFull := a_pBufferZoneChildSIF[usiNumOfBufferZones-1]^.Cur.bolBufferFull;	
	// All buffers full -> based on all zones
	SIf.Cur.bolAllBuffersFull:= THIS^.checkAllZonesFull();
	// Approximate number of hangers in buffer -> based on all zones
	SIf.Cur.dinNumOfHangersInBuffer:= THIS^.CalcSumNumOfHangers();
	// Max. buffer capacity -> based on all zones
	SIf.Cur.dinMaxCapacity:= THIS^.CalcMaxCapacity();	
	// Hangers passed total counter, always from zone 1, output
	SIf.Cur.dinHangersPassedTotal:= a_pBufferZoneChildSIF[0]^.Cur.dinHangersPassedTotal;
	// Hanger detected, always from zone 1, output
	SIf.Cur.bolHangerDetected:= a_pBufferZoneChildSIF[0]^.Cur.bolHangerDetected;
	// Number of passing hangers per pulse in first zone
	SIf.Cur.uinNumOfHangersPerPulseFirstZone:= a_pBufferZoneChildSIF[0]^.Cfg.uinNumOfHangersPerPulse;
	
	
	// Set alarm all buffer zones full
	IF (SIf.Cur.bolAllBuffersFull = TRUE) THEN	
		// SIf.Alm[3].strText := 'All buffer zones full';	 
		pfbAlarmCtrl^.setAlarm(CIf.Info.intCtrlId,3,0,ADR(SIf.Alm),E_AlmState.RST,CIf.Job.eMe_ActivAlmClass);	
	END_IF
			
END_IF

// ----------------------------------------------------------------------------------
// Conditions Always
// overrule error always from base -> no EOFF State!! in EOFF go to OFF
IF (me.StateMachine.intStateNext = cSTA_EOFFBusy) THEN
	IF (me.StateMachine.intState=cSTA_OFF) THEN
		me.StateMachine.intStateNext := cSTA_OFF;
	ELSE // stay in OFF
		me.StateMachine.intStateNext := cSTA_OFFBusy;
	END_IF
END_IF
END_METHOD

PROPERTY BufferFull : BOOL
GET
BufferFull:= SIf.Cur.bolAllBuffersFull;
END_GET
END_PROPERTY

METHOD PROTECTED CalcMaxCapacity : DINT
VAR
	ii: INT;
	dinSumMaxCapacity: DINT;
END_VAR
// Method calculate the sum of max. capacities in all zones and return the result.

//Init
CalcMaxCapacity:= 0;
dinSumMaxCapacity:= 0;

// Loop over all childs
FOR ii:=0 TO usiNumOfBufferZones-1 BY 1 DO
	// Build sum of all zones		
	dinSumMaxCapacity:= dinSumMaxCapacity + a_pBufferZoneChildSIF[ii]^.Cfg.dinMaxCapacity; 	
END_FOR

// Return result
CalcMaxCapacity:= dinSumMaxCapacity;
END_METHOD

METHOD PROTECTED CalcSumNumOfHangers : DINT
VAR
	ii: INT;
	dinSumNumOfHangers: DINT;
END_VAR
// Method calculate the sum of hangers in all zones and return the result.

//Init
CalcSumNumOfHangers:= 0;
dinSumNumOfHangers:= 0;

// Loop over all childs
FOR ii:=0 TO usiNumOfBufferZones-1 BY 1 DO
	// Build sum of all zones		
	dinSumNumOfHangers:= dinSumNumOfHangers + a_pBufferZoneChildSIF[ii]^.Cur.dinNumOfHangersInBuffer; 	
END_FOR

// Return result
CalcSumNumOfHangers:= dinSumNumOfHangers;
END_METHOD

METHOD PROTECTED checkAllZonesEmpty : BOOL
VAR
	ii: INT;
	usiNumOfEmptyZones: USINT;
END_VAR
// Method check if all zones are empty. If yes, return TRUE

//Init
checkAllZonesEmpty:= FALSE;
usiNumOfEmptyZones:= 0;

// Loop over all childs
FOR ii:=0 TO usiNumOfBufferZones-1 BY 1 DO
	// Check number of hangers in buffer zone X <= 0	
	IF (a_pBufferZoneChildSIF[ii]^.Cur.dinNumOfHangersInBuffer <= 0) THEN
		usiNumOfEmptyZones:= usiNumOfEmptyZones+1;		
	END_IF
END_FOR

// All zones empty
IF (usiNumOfEmptyZones = usiNumOfBufferZones) THEN
	checkAllZonesEmpty:= TRUE;
END_IF
END_METHOD

METHOD PROTECTED checkAllZonesFull : BOOL
VAR
	ii: INT;
	usiNumOfFullZones: USINT;
END_VAR
// Method check if all zones are full. If yes, return TRUE

//Init
checkAllZonesFull:= FALSE;
usiNumOfFullZones:= 0;

// Loop over all childs
FOR ii:=0 TO usiNumOfBufferZones-1 BY 1 DO
	// Check buffer full info of zone X	
	IF (a_pBufferZoneChildSIF[ii]^.Cur.bolBufferFull=TRUE) THEN
		usiNumOfFullZones:= usiNumOfFullZones+1;		
	END_IF
END_FOR

// All zones full
IF (usiNumOfFullZones = usiNumOfBufferZones) THEN
	checkAllZonesFull:= TRUE;
END_IF
END_METHOD

METHOD checkChildAlmClass : BOOL
//------------------------------------------------------------------------------------------------------
// check child alarm classes
// set me alarm class active if at least one child has an EOFF
IF CheckAllChildAlmClass(E_AlmClass.EOFF) THEN
	CIf.Job.eMe_ActivAlmClass := E_AlmClass.EOFF;
	me.Alarm.bolfp := TRUE;
ELSIF CheckAllChildAlmClass(E_AlmClass.OFF) THEN
	CIf.Job.eMe_ActivAlmClass := E_AlmClass.OFF;
	me.Alarm.bolfp := TRUE;
ELSIF CheckAllChildAlmClass(E_AlmClass.STOP) THEN // FB_SLB needs alarm class STOP
	CIf.Job.eMe_ActivAlmClass := E_AlmClass.STOP;
	me.Alarm.bolfp := TRUE;
ELSE
	IF (me.Alarm.bolfp) THEN
		CIf.Job.eMe_ActivAlmClass := E_AlmClass.NONE; // no reset necessary
		me.Alarm.bolfp := FALSE;
	END_IF
END_IF

